PROGRAM MAIN
VAR
	instFB_DryingSectionLubrificationControl_V1 : FB_DryingSectionLubrificationControl_V1;
	instFB_SavePersistentData	: FB_SavePersistentData;
	instFB_SpeedDroopControlMst : FB_SpeedDroopControl_1;
	instFB_SpeedDroopControlSlv : FB_FormingBoardDriveControl;
	instFB_DryingSectionDriveControl_GR1 : FB_DryingSectionDriveControl_V1;
	instFB_DryingSectionDriveControl_GR2 : FB_DryingSectionDriveControl_V1;
	
	instFFB_PressSectionDriveControl_V1 : FB_PressSectionDriveControl_V2;

	                 

	FB_SoftstarterWithBypass_0: FB_SoftstarterWithBypass;
	FB_PressureControl_0: FB_PressureControl;
	FB_MixPumpControl_0: FB_MixPumpControl;
	FB_HeadboxLipsPWMControl_0: FB_HeadboxLipsPWMControl;
	instPWM: CTRL_PWM;
	instFB_MixPumpControl: FB_MixPumpControl;
	instFB_FormingBoardRollUpDown: FB_FormingBoardRollUpDown;
	instFB_HeadboxLipsPWMControl: FB_HeadboxLipsPWMControl;
	instFB_FormingBoarWireStrech: FB_FormingBoardRollUpDown;
	instFB_FormingBoardWireStretchControl: FB_FormingBoardWireStretchControl;
	instFB_SoftstarterSimpleCPS: FB_SimpleMotorStart_V2;
	// Centrifugal Pressure Screen (CPS) running (Depurador cabeçeira)
	CPSRunning: BOOL;
	instFB_LevelControlWirePit: FB_LevelControl_V2;
	instFB_LevelControlCouchPit: FB_LevelControl_V2;
	stop: BOOL;
	formingBoardWireLimitInibit: BOOL;
	instFB_SoftstarterSimpleCouchPitMixer: FB_SimpleMotorStart_V2;
	instFB_SoftstarterWithBypassFormingBoard: FB_SoftstarterWithBypass;
	instFB_SoftstarterWithBypassSuctionRoll: FB_SoftstarterWithBypass_V1;
	FB_SoftstarterWithBypassTest: FB_SoftstarterWithBypass;
	FB_SimpleMotorStart_V2_Test: FB_SimpleMotorStart_V2;
	instFB_SoftstarterWithBypass_V1: FB_SoftstarterWithBypass_V1;
	instFB_PressureControl_V1StockPumpC: FB_PressureControl_V1;
	instFB_SoftstarterWithBypass_FormingBoard: FB_SoftstarterWithBypass_V1;
	instFB_PressureControl_V1: FB_PressureControl_V1;
	instFB_FormingBoardDriveControl_V1: FB_FormingBoardControl_V1;
	instFB_MixPumpControl_V1: FB_MixPumpControl_V1;
	instFB_ProcessControlerStockPump: FB_ProcessControler;
	instFB_ProcessControlerWirePitPump: FB_ProcessControler;
	
	formingBoardNextGrReference: REAL;
	pressSectionNextGrReference: REAL;
	dryingSec1NextGrReference: REAL;
	dryingSec2NextGrReference: REAL;
	
	instFB_DryingSectionDriveControl_GR3: FB_DryingSectionDriveControl_V1;
	
	instFB_DryingSectionDriveControlV2_GR3: FB_DryingSectionDriveControl_V2;
	
	
	
	instFB_RewinderControl_V1 : FB_RewinderControl_V1;
	
	
	
	instFB_DryingSectionDriveControl_V3_GR1: FB_DryingSectionDriveControl_V3;
	instFB_DryingSectionDriveControl_V3_GR2: FB_DryingSectionDriveControl_V3;
	instFB_DryingSectionDriveControl_V3_GR3: FB_DryingSectionDriveControl_V3;
	
	
	initVariables : BOOL;
	rInitVariables : BOOL;
	initVariablesOld : BOOL;
	
	
	dryingSectionGr1NextGroupReference: REAL;
	dryingSectionGr2NextGroupReference: REAL;
	dryingSectionGr3NextGroupReference: REAL;
	instFB_SoftstarterWithBypassPress1: FB_SoftstarterWithBypass_V1;
	instFB_SoftstarterWithBypassPress2: FB_SoftstarterWithBypass_V1;
	bypassFault: BOOL;
	startNotAllowed: BOOL;
	instFB_WinderDriveControl_V1: FB_WinderDriveControl_V1;
	FB_FormingBoardControl_V3_0: FB_FormingBoardControl_V3;
	pressSectionNextGroupReference: REAL;
	
	
	firstScan	:BOOL := TRUE;
	
	
	vacumPumpSoftStartOK: BOOL;
	instTOFvacumPumpSoftstart: TOF;
	startSoftstartContactorFromPressFelt1: BOOL;
	startSoftstartFromPressFelt1: BOOL;
	startSoftstartContactorFromPressFelt2: BOOL;
	startSoftstartFromPressFelt2: BOOL;
	instFB_FB_SimpleMotorStart_V3_VaccumSealPump: FB_SimpleMotorStart_V3;
	instFB_FB_SimpleMotorStart_V3_lowVacuumExhaustFan: FB_SimpleMotorStart_V3;
	instFB_FB_SimpleMotorStart_V3_VaccumSeparator: FB_SimpleMotorStart_V3;
	instFB_FB_SimpleMotorStart_V3_FormingTailCutterNozzle: FB_SimpleMotorStart_V3;
	instFB_FB_SimpleMotorStart_V3_FormingWireShower: FB_SimpleMotorStart_V3;
	
	instFB_AlarmControl	: FB_AlarmControl;
	
END_VAR

//────────────────────────────────────────────
// READ I/O MODULES
//────────────────────────────────────────────

// UG I/O Modules
P1_100_UG01();
P1_100_UG02();
P1_100_UG03_SuctionRoll();
P1_100_UG04();
P1_100_UG05();
P1_300_UG06_TractionRoll();

// Digital Inputs
P1_050_DI1();
P1_050_DI2();
P1_050_DI3();
P9_050_DI1();
P9_050_DI2();
P9_050_DI3();
P10_050_DI1();
P10_050_DI2();
P10_050_DI3();
P10_050_DI4();
P10_050_DI5();
P10_050_DI6();
P10_050_DI7();
P10_050_DI8();

// Digital Outputs
P1_050_DO1();
P1_050_DO2();
P1_050_DO3();
P9_050_DO1();
P9_050_DO2();
P9_050_DO3();
P10_050_DO1();
P10_050_DO2();
P10_050_DO3();
P10_050_DO4();

// Analog Inputs
P1_050_AI1();
P1_050_AI2();
P1_050_AI3();
P1_050_AI4();
P9_050_AI1();
P10_050_AI1();
P10_050_AI2();

// Analog Outputs
P1_050_AQ1();
P1_050_AQ2();
P10_050_AO1();


CP1_050_DI1();
CP1_050_DO1();
CP1_050_AO1();


// Safety PLC
P1_050_SP1();

//────────────────────────────────────────────
// READ DRIVES
//────────────────────────────────────────────

// Press Section
P11_400_UG01_SecondPress();     // Second Press
P12_400_UG01_FirstPress();      // First Press

// Drying Section — Group 1
P13_500_UG01_1GR_UpperSlave();  // Group 1 - Upper Slave
P13_500_UG02_1GR_LowerMaster(); // Group 1 - Lower Master
P13_500_UG03_1GR_UpperMaster(); // Group 1 - Upper Master

// Drying Section — Group 2
P13_501_UG01_2GR_LowerSlave();  // Group 2 - Lower Slave
P13_501_UG02_2GR_UpperSlave();  // Group 2 - Upper Slave
P13_501_UG03_2GR_LowerMaster(); // Group 2 - Lower Master
P14_501_UG01_2GR_UpperMaster(); // Group 2 - Upper Master

// Drying Section — Group 3
P14_502_UG01_3GR_LowerSlave();  // Group 3 - Lower Slave
P14_502_UG02_3GR_UpperSlave();  // Group 3 - Upper Slave
P14_502_UG03_3GR_LowerMaster(); // Group 3 - Lower Master
P14_502_UG04_3GR_UpperMaster(); // Group 3 - Upper Master

//Winder group
P15_600_UG01_Rewinder();
//────────────────────────────────────────────
// PROGRAM FUNCTION BLOCK CALLS
//────────────────────────────────────────────

// Forming Section
_100_FormingBoardControl();
_110_FormingBoardAux();

// Press Section
_200_PressSectionControl();

// Drying Section
_500_DryingSectionGroup1DriveControl();
_501_DryingSectionGroup2DriveControl();
_502_DryingSectionGroup3DriveControl();
_550_DryingSectionLubrification();
_600_WinderGroup();

_888_Alarms();


// Headbox / Stock Prep / Wet End Auxiliary Systems
//_HeadBoxAuxiliaryControls();
_MixPumpControl_1();
_WirePitPumpControl_1();
_CentrifugalPressureScreenControl();
_CouchPitPumpControl();
_CouchPitMixerControl();
_VaccumPumps();
//_StockPumpControl();
_StockPumpControl_1();

// Testing & Debug
_FunctionBlockTest();

//────────────────────────────────────────────
// SYSTEM MANAGEMENT
//────────────────────────────────────────────

// Save persistent variables to CPU
instFB_SavePersistentData();

// Enable Safety PLC
P1_050_SP1.run := TRUE;

// Perform machine-wide reset
machineReset();


rInitVariables := initVariables AND NOT initVariablesOld;

IF rInitVariables THEN
	
	_000_Init_Variables();

END_IF

initVariablesOld := initVariables;



IF firstScan THEN
	
	_001_FirstScan();

END_IF

METHOD _000_Init_Variables
VAR_INPUT
END_VAR

P1_300_UG06_TractionRoll.deviceConfig.MotorSpeedInputLow := 0.0;
P1_300_UG06_TractionRoll.deviceConfig.MotorSpeedInputHigh := 360.4;
P1_300_UG06_TractionRoll.deviceConfig.MotorSpeedOutputLow := 0.0;
P1_300_UG06_TractionRoll.deviceConfig.MotorSpeedOutputHigh := 360.4;
P1_300_UG06_TractionRoll.deviceConfig.speedSetpointInputLow := 0.0;
P1_300_UG06_TractionRoll.deviceConfig.speedSetpointInputHigh := 360.4;
P1_300_UG06_TractionRoll.deviceConfig.speedSetpointOutputLow := 0.0;
P1_300_UG06_TractionRoll.deviceConfig.speedSetpointOutputHigh := 360.4;


P1_100_UG03_SuctionRoll.deviceConfig.MotorSpeedInputLow := 0.0;
P1_100_UG03_SuctionRoll.deviceConfig.MotorSpeedInputHigh := 329.3;
P1_100_UG03_SuctionRoll.deviceConfig.MotorSpeedOutputLow := 0.0;
P1_100_UG03_SuctionRoll.deviceConfig.MotorSpeedOutputHigh := 329.3;
P1_100_UG03_SuctionRoll.deviceConfig.speedSetpointInputLow := 0.0;
P1_100_UG03_SuctionRoll.deviceConfig.speedSetpointInputHigh := 329.3;
P1_100_UG03_SuctionRoll.deviceConfig.speedSetpointOutputLow := 0.0;
P1_100_UG03_SuctionRoll.deviceConfig.speedSetpointOutputHigh := 329.3;
//Torque Enable
P1_100_UG03_SuctionRoll.deviceConfig.torqueLimiterEnabled := TRUE;
P1_100_UG03_SuctionRoll.deviceConfig.operationMode := 4;



P11_400_UG01_SecondPress.deviceConfig.MotorSpeedInputLow := 0.0;
P11_400_UG01_SecondPress.deviceConfig.MotorSpeedInputHigh := 374;
P11_400_UG01_SecondPress.deviceConfig.MotorSpeedOutputLow := 0.0;
P11_400_UG01_SecondPress.deviceConfig.MotorSpeedOutputHigh := 374;
P11_400_UG01_SecondPress.deviceConfig.speedSetpointInputLow := 0.0;
P11_400_UG01_SecondPress.deviceConfig.speedSetpointInputHigh := 374;
P11_400_UG01_SecondPress.deviceConfig.speedSetpointOutputLow := 0.0;
P11_400_UG01_SecondPress.deviceConfig.speedSetpointOutputHigh := 374;


P12_400_UG01_FirstPress.deviceConfig.MotorSpeedInputLow := 0.0;
P12_400_UG01_FirstPress.deviceConfig.MotorSpeedInputHigh := 239.9;
P12_400_UG01_FirstPress.deviceConfig.MotorSpeedOutputLow := 0.0;
P12_400_UG01_FirstPress.deviceConfig.MotorSpeedOutputHigh := 239.9;
P12_400_UG01_FirstPress.deviceConfig.speedSetpointInputLow := 0.0;
P12_400_UG01_FirstPress.deviceConfig.speedSetpointInputHigh := 239.9;
P12_400_UG01_FirstPress.deviceConfig.speedSetpointOutputLow := 0.0;
P12_400_UG01_FirstPress.deviceConfig.speedSetpointOutputHigh := 239.9;
//Torque Enable
P12_400_UG01_FirstPress.deviceConfig.torqueLimiterEnabled := TRUE;
P12_400_UG01_FirstPress.deviceConfig.operationMode := 4;



//============================
// DRYING SECTION — GROUP 1
//============================

// Upper Slave
P13_500_UG01_1GR_UpperSlave.deviceConfig.MotorSpeedInputLow := 0.0;
P13_500_UG01_1GR_UpperSlave.deviceConfig.MotorSpeedInputHigh := 750;
P13_500_UG01_1GR_UpperSlave.deviceConfig.MotorSpeedOutputLow := 0.0;
P13_500_UG01_1GR_UpperSlave.deviceConfig.MotorSpeedOutputHigh := 750;
P13_500_UG01_1GR_UpperSlave.deviceConfig.speedSetpointInputLow := 0.0;
P13_500_UG01_1GR_UpperSlave.deviceConfig.speedSetpointInputHigh := 750;
P13_500_UG01_1GR_UpperSlave.deviceConfig.speedSetpointOutputLow := 0.0;
P13_500_UG01_1GR_UpperSlave.deviceConfig.speedSetpointOutputHigh := 750;
P13_500_UG01_1GR_UpperSlave.deviceConfig.torqueLimiterEnabled := TRUE;
P13_500_UG01_1GR_UpperSlave.deviceConfig.operationMode := 4;

// Lower Master
P13_500_UG02_1GR_LowerMaster.deviceConfig.MotorSpeedInputLow := 0.0;
P13_500_UG02_1GR_LowerMaster.deviceConfig.MotorSpeedInputHigh := 750;
P13_500_UG02_1GR_LowerMaster.deviceConfig.MotorSpeedOutputLow := 0.0;
P13_500_UG02_1GR_LowerMaster.deviceConfig.MotorSpeedOutputHigh := 750;
P13_500_UG02_1GR_LowerMaster.deviceConfig.speedSetpointInputLow := 0.0;
P13_500_UG02_1GR_LowerMaster.deviceConfig.speedSetpointInputHigh := 750;
P13_500_UG02_1GR_LowerMaster.deviceConfig.speedSetpointOutputLow := 0.0;
P13_500_UG02_1GR_LowerMaster.deviceConfig.speedSetpointOutputHigh := 750;
//P13_500_UG02_1GR_LowerMaster.deviceConfig.torqueLimiterEnabled := FALSE;
//P13_500_UG02_1GR_LowerMaster.deviceConfig.operationMode := 4;

// Upper Master
P13_500_UG03_1GR_UpperMaster.deviceConfig.MotorSpeedInputLow := 0.0;
P13_500_UG03_1GR_UpperMaster.deviceConfig.MotorSpeedInputHigh := 750;
P13_500_UG03_1GR_UpperMaster.deviceConfig.MotorSpeedOutputLow := 0.0;
P13_500_UG03_1GR_UpperMaster.deviceConfig.MotorSpeedOutputHigh := 750;
P13_500_UG03_1GR_UpperMaster.deviceConfig.speedSetpointInputLow := 0.0;
P13_500_UG03_1GR_UpperMaster.deviceConfig.speedSetpointInputHigh := 750;
P13_500_UG03_1GR_UpperMaster.deviceConfig.speedSetpointOutputLow := 0.0;
P13_500_UG03_1GR_UpperMaster.deviceConfig.speedSetpointOutputHigh := 750;
//P13_500_UG03_1GR_UpperMaster.deviceConfig.torqueLimiterEnabled := FALSE;
//P13_500_UG03_1GR_UpperMaster.deviceConfig.operationMode := 4;


//============================
// DRYING SECTION — GROUP 2
//============================

// Lower Slave
P13_501_UG01_2GR_LowerSlave.deviceConfig.MotorSpeedInputLow := 0.0;
P13_501_UG01_2GR_LowerSlave.deviceConfig.MotorSpeedInputHigh := 750;
P13_501_UG01_2GR_LowerSlave.deviceConfig.MotorSpeedOutputLow := 0.0;
P13_501_UG01_2GR_LowerSlave.deviceConfig.MotorSpeedOutputHigh := 750;
P13_501_UG01_2GR_LowerSlave.deviceConfig.speedSetpointInputLow := 0.0;
P13_501_UG01_2GR_LowerSlave.deviceConfig.speedSetpointInputHigh := 750;
P13_501_UG01_2GR_LowerSlave.deviceConfig.speedSetpointOutputLow := 0.0;
P13_501_UG01_2GR_LowerSlave.deviceConfig.speedSetpointOutputHigh := 750;
P13_501_UG01_2GR_LowerSlave.deviceConfig.torqueLimiterEnabled := TRUE;
P13_501_UG01_2GR_LowerSlave.deviceConfig.operationMode := 4;

// Upper Slave
P13_501_UG02_2GR_UpperSlave.deviceConfig.MotorSpeedInputLow := 0.0;
P13_501_UG02_2GR_UpperSlave.deviceConfig.MotorSpeedInputHigh := 750;
P13_501_UG02_2GR_UpperSlave.deviceConfig.MotorSpeedOutputLow := 0.0;
P13_501_UG02_2GR_UpperSlave.deviceConfig.MotorSpeedOutputHigh := 750;
P13_501_UG02_2GR_UpperSlave.deviceConfig.speedSetpointInputLow := 0.0;
P13_501_UG02_2GR_UpperSlave.deviceConfig.speedSetpointInputHigh := 750;
P13_501_UG02_2GR_UpperSlave.deviceConfig.speedSetpointOutputLow := 0.0;
P13_501_UG02_2GR_UpperSlave.deviceConfig.speedSetpointOutputHigh := 750;
P13_501_UG02_2GR_UpperSlave.deviceConfig.torqueLimiterEnabled := TRUE;
P13_501_UG02_2GR_UpperSlave.deviceConfig.operationMode := 4;

// Lower Master
P13_501_UG03_2GR_LowerMaster.deviceConfig.MotorSpeedInputLow := 0.0;
P13_501_UG03_2GR_LowerMaster.deviceConfig.MotorSpeedInputHigh := 750;
P13_501_UG03_2GR_LowerMaster.deviceConfig.MotorSpeedOutputLow := 0.0;
P13_501_UG03_2GR_LowerMaster.deviceConfig.MotorSpeedOutputHigh := 750;
P13_501_UG03_2GR_LowerMaster.deviceConfig.speedSetpointInputLow := 0.0;
P13_501_UG03_2GR_LowerMaster.deviceConfig.speedSetpointInputHigh := 750;
P13_501_UG03_2GR_LowerMaster.deviceConfig.speedSetpointOutputLow := 0.0;
P13_501_UG03_2GR_LowerMaster.deviceConfig.speedSetpointOutputHigh := 750;
//P13_501_UG03_2GR_LowerMaster.deviceConfig.torqueLimiterEnabled := FALSE;
//P13_501_UG03_2GR_LowerMaster.deviceConfig.operationMode := 4;

// Upper Master
P14_501_UG01_2GR_UpperMaster.deviceConfig.MotorSpeedInputLow := 0.0;
P14_501_UG01_2GR_UpperMaster.deviceConfig.MotorSpeedInputHigh := 750;
P14_501_UG01_2GR_UpperMaster.deviceConfig.MotorSpeedOutputLow := 0.0;
P14_501_UG01_2GR_UpperMaster.deviceConfig.MotorSpeedOutputHigh := 750;
P14_501_UG01_2GR_UpperMaster.deviceConfig.speedSetpointInputLow := 0.0;
P14_501_UG01_2GR_UpperMaster.deviceConfig.speedSetpointInputHigh := 750;
P14_501_UG01_2GR_UpperMaster.deviceConfig.speedSetpointOutputLow := 0.0;
P14_501_UG01_2GR_UpperMaster.deviceConfig.speedSetpointOutputHigh := 750;
//P14_501_UG01_2GR_UpperMaster.deviceConfig.torqueLimiterEnabled := FALSE;
//P14_501_UG01_2GR_UpperMaster.deviceConfig.operationMode := 4;


//============================
// DRYING SECTION — GROUP 3
//============================

// Lower Slave
P14_502_UG01_3GR_LowerSlave.deviceConfig.MotorSpeedInputLow := 0.0;
P14_502_UG01_3GR_LowerSlave.deviceConfig.MotorSpeedInputHigh := 750;
P14_502_UG01_3GR_LowerSlave.deviceConfig.MotorSpeedOutputLow := 0.0;
P14_502_UG01_3GR_LowerSlave.deviceConfig.MotorSpeedOutputHigh := 750;
P14_502_UG01_3GR_LowerSlave.deviceConfig.speedSetpointInputLow := 0.0;
P14_502_UG01_3GR_LowerSlave.deviceConfig.speedSetpointInputHigh := 750;
P14_502_UG01_3GR_LowerSlave.deviceConfig.speedSetpointOutputLow := 0.0;
P14_502_UG01_3GR_LowerSlave.deviceConfig.speedSetpointOutputHigh := 750;
P14_502_UG01_3GR_LowerSlave.deviceConfig.torqueLimiterEnabled := TRUE;
P14_502_UG01_3GR_LowerSlave.deviceConfig.operationMode := 4;

// Upper Slave
P14_502_UG02_3GR_UpperSlave.deviceConfig.MotorSpeedInputLow := 0.0;
P14_502_UG02_3GR_UpperSlave.deviceConfig.MotorSpeedInputHigh := 750;
P14_502_UG02_3GR_UpperSlave.deviceConfig.MotorSpeedOutputLow := 0.0;
P14_502_UG02_3GR_UpperSlave.deviceConfig.MotorSpeedOutputHigh := 750;
P14_502_UG02_3GR_UpperSlave.deviceConfig.speedSetpointInputLow := 0.0;
P14_502_UG02_3GR_UpperSlave.deviceConfig.speedSetpointInputHigh := 750;
P14_502_UG02_3GR_UpperSlave.deviceConfig.speedSetpointOutputLow := 0.0;
P14_502_UG02_3GR_UpperSlave.deviceConfig.speedSetpointOutputHigh := 750;
P14_502_UG02_3GR_UpperSlave.deviceConfig.torqueLimiterEnabled := TRUE;
P14_502_UG02_3GR_UpperSlave.deviceConfig.operationMode := 4;

// Lower Master
P14_502_UG03_3GR_LowerMaster.deviceConfig.MotorSpeedInputLow := 0.0;
P14_502_UG03_3GR_LowerMaster.deviceConfig.MotorSpeedInputHigh := 750;
P14_502_UG03_3GR_LowerMaster.deviceConfig.MotorSpeedOutputLow := 0.0;
P14_502_UG03_3GR_LowerMaster.deviceConfig.MotorSpeedOutputHigh := 750;
P14_502_UG03_3GR_LowerMaster.deviceConfig.speedSetpointInputLow := 0.0;
P14_502_UG03_3GR_LowerMaster.deviceConfig.speedSetpointInputHigh := 750;
P14_502_UG03_3GR_LowerMaster.deviceConfig.speedSetpointOutputLow := 0.0;
P14_502_UG03_3GR_LowerMaster.deviceConfig.speedSetpointOutputHigh := 750;
//P14_502_UG03_3GR_LowerMaster.deviceConfig.torqueLimiterEnabled := FALSE;
//P14_502_UG03_3GR_LowerMaster.deviceConfig.operationMode := 4;

// Upper Master
P14_502_UG04_3GR_UpperMaster.deviceConfig.MotorSpeedInputLow := 0.0;
P14_502_UG04_3GR_UpperMaster.deviceConfig.MotorSpeedInputHigh := 750;
P14_502_UG04_3GR_UpperMaster.deviceConfig.MotorSpeedOutputLow := 0.0;
P14_502_UG04_3GR_UpperMaster.deviceConfig.MotorSpeedOutputHigh := 750;
P14_502_UG04_3GR_UpperMaster.deviceConfig.speedSetpointInputLow := 0.0;
P14_502_UG04_3GR_UpperMaster.deviceConfig.speedSetpointInputHigh := 750;
P14_502_UG04_3GR_UpperMaster.deviceConfig.speedSetpointOutputLow := 0.0;
P14_502_UG04_3GR_UpperMaster.deviceConfig.speedSetpointOutputHigh := 750;
//P14_502_UG04_3GR_UpperMaster.deviceConfig.torqueLimiterEnabled := FALSE;
//P14_502_UG04_3GR_UpperMaster.deviceConfig.operationMode := 4;
END_METHOD

METHOD _001_FirstScan
VAR_INPUT
END_VAR

(*

paperMachineHmiCommands.dryingSectionGroup1SteamPressureAutoMan := FALSE;

	dryingSectionGroup1SteamPressureAutoSetpoint : REAL;  // Recovery speed increment [m/min or %] (Incremento de recuperação Grupo 1)
	dryingSectionGroup1SteamPressureManualSetpoint : REAL;  // Recovery speed increment [m/min or %] (Incremento de recuperação Grupo 1)
	
*)



paperMachineHmiCommands.dryingSectionGroup1SteamPressureAutoMan := FALSE;
paperMachineHmiCommands.dryingSectionGroup1SteamPressureManualSetpoint := 0.0;

paperMachineHmiCommands.dryingSectionGroup2SteamPressureAutoMan := FALSE;
paperMachineHmiCommands.dryingSectionGroup2SteamPressureManualSetpoint := 0.0;

paperMachineHmiCommands.dryingSectionGroup3SteamPressureAutoMan := FALSE;
paperMachineHmiCommands.dryingSectionGroup3SteamPressureManualSetpoint := 0.0;


//Reset first scan flag
firstScan := FALSE;
END_METHOD

METHOD _100_FormingBoardControl
VAR_INPUT
END_VAR
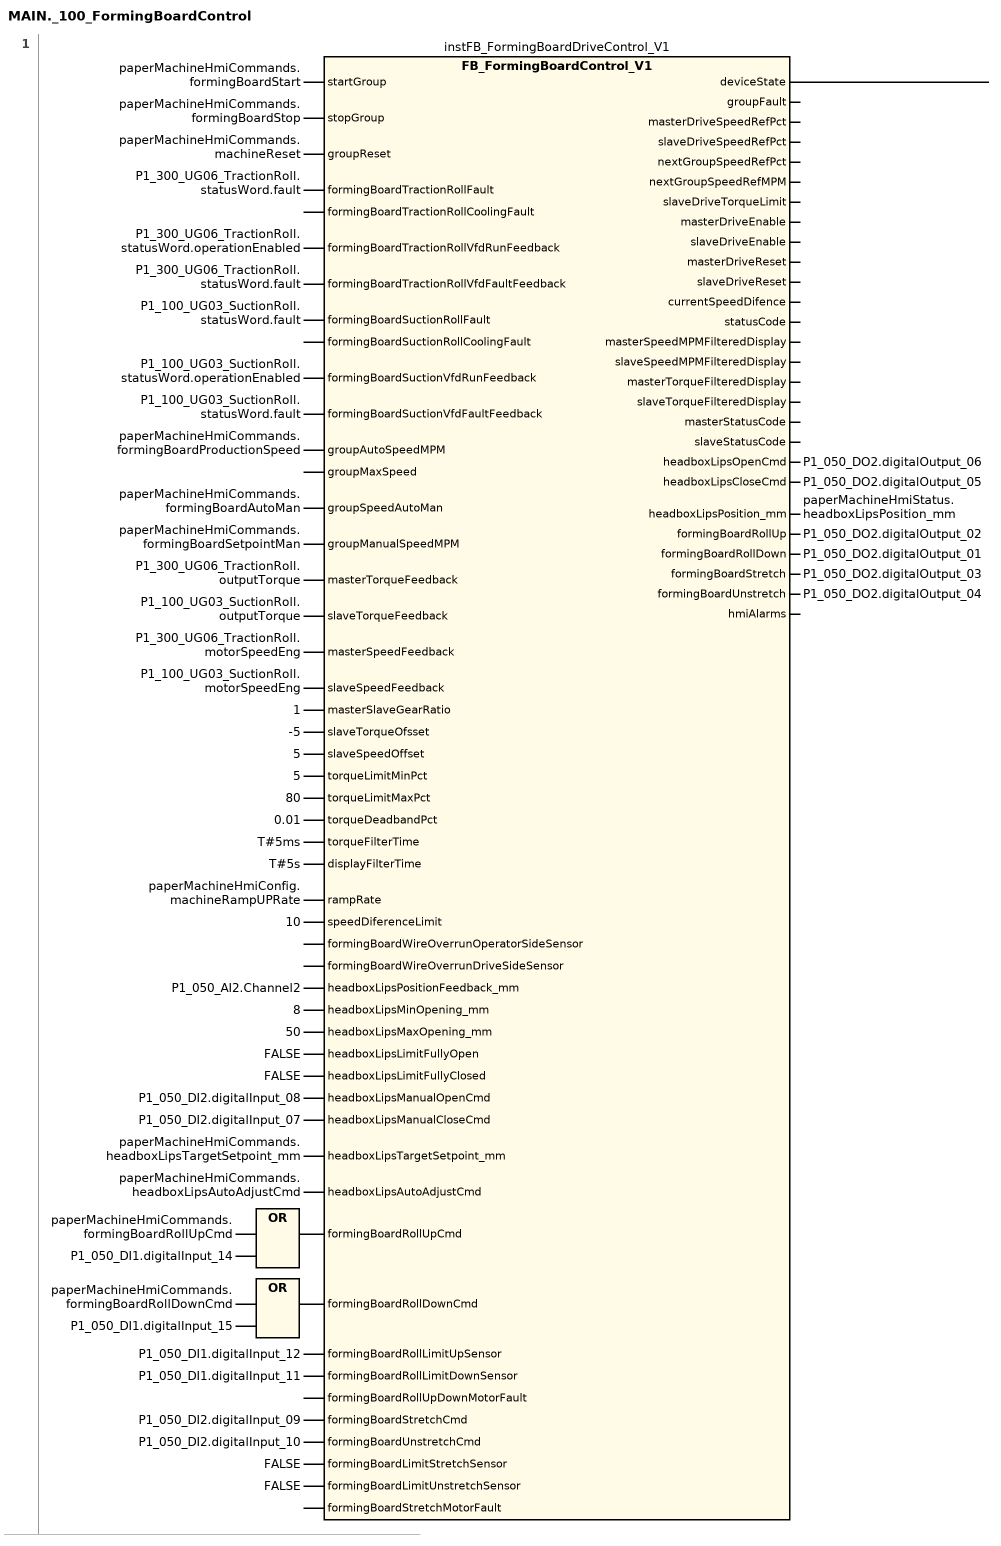
// NETWORK 1
instFB_FormingBoardDriveControl_V1(
    startGroup := paperMachineHmiCommands.formingBoardStart,
    stopGroup := paperMachineHmiCommands.formingBoardStop,
    groupReset := paperMachineHmiCommands.machineReset,
    formingBoardTractionRollFault := P1_300_UG06_TractionRoll.statusWord.fault,
    formingBoardTractionRollVfdRunFeedback := P1_300_UG06_TractionRoll.statusWord.operationEnabled,
    formingBoardTractionRollVfdFaultFeedback := P1_300_UG06_TractionRoll.statusWord.fault,
    formingBoardSuctionRollFault := P1_100_UG03_SuctionRoll.statusWord.fault,
    formingBoardSuctionVfdRunFeedback := P1_100_UG03_SuctionRoll.statusWord.operationEnabled,
    formingBoardSuctionVfdFaultFeedback := P1_100_UG03_SuctionRoll.statusWord.fault,
    groupAutoSpeedMPM := paperMachineHmiCommands.formingBoardProductionSpeed,
    groupSpeedAutoMan := paperMachineHmiCommands.formingBoardAutoMan,
    groupManualSpeedMPM := paperMachineHmiCommands.formingBoardSetpointMan,
    masterTorqueFeedback := P1_300_UG06_TractionRoll.outputTorque,
    slaveTorqueFeedback := P1_100_UG03_SuctionRoll.outputTorque,
    masterSpeedFeedback := P1_300_UG06_TractionRoll.motorSpeedEng,
    slaveSpeedFeedback := P1_100_UG03_SuctionRoll.motorSpeedEng,
    masterSlaveGearRatio := 1,
    slaveTorqueOfsset := -5,
    slaveSpeedOffset := 5,
    torqueLimitMinPct := 5,
    torqueLimitMaxPct := 80,
    torqueDeadbandPct := 0.01,
    torqueFilterTime := T#5ms,
    displayFilterTime := T#5s,
    rampRate := paperMachineHmiConfig.machineRampUPRate,
    speedDiferenceLimit := 10,
    headboxLipsPositionFeedback_mm := P1_050_AI2.Channel2,
    headboxLipsMinOpening_mm := 8,
    headboxLipsMaxOpening_mm := 50,
    headboxLipsLimitFullyOpen := FALSE,
    headboxLipsLimitFullyClosed := FALSE,
    headboxLipsManualOpenCmd := P1_050_DI2.digitalInput_08,
    headboxLipsManualCloseCmd := P1_050_DI2.digitalInput_07,
    headboxLipsTargetSetpoint_mm := paperMachineHmiCommands.headboxLipsTargetSetpoint_mm,
    headboxLipsAutoAdjustCmd := paperMachineHmiCommands.headboxLipsAutoAdjustCmd,
    formingBoardRollUpCmd := paperMachineHmiCommands.formingBoardRollUpCmd OR P1_050_DI1.digitalInput_14,
    formingBoardRollDownCmd := paperMachineHmiCommands.formingBoardRollDownCmd OR P1_050_DI1.digitalInput_15,
    formingBoardRollLimitUpSensor := P1_050_DI1.digitalInput_12,
    formingBoardRollLimitDownSensor := P1_050_DI1.digitalInput_11,
    formingBoardStretchCmd := P1_050_DI2.digitalInput_09,
    formingBoardUnstretchCmd := P1_050_DI2.digitalInput_10,
    formingBoardLimitStretchSensor := FALSE,
    formingBoardLimitUnstretchSensor := FALSE,
    headboxLipsOpenCmd => P1_050_DO2.digitalOutput_06,
    headboxLipsCloseCmd => P1_050_DO2.digitalOutput_05,
    headboxLipsPosition_mm => paperMachineHmiStatus.headboxLipsPosition_mm,
    formingBoardRollUp => P1_050_DO2.digitalOutput_02,
    formingBoardRollDown => P1_050_DO2.digitalOutput_01,
    formingBoardStretch => P1_050_DO2.digitalOutput_03,
    formingBoardUnstretch => P1_050_DO2.digitalOutput_04); // FB_FormingBoardControl_V1

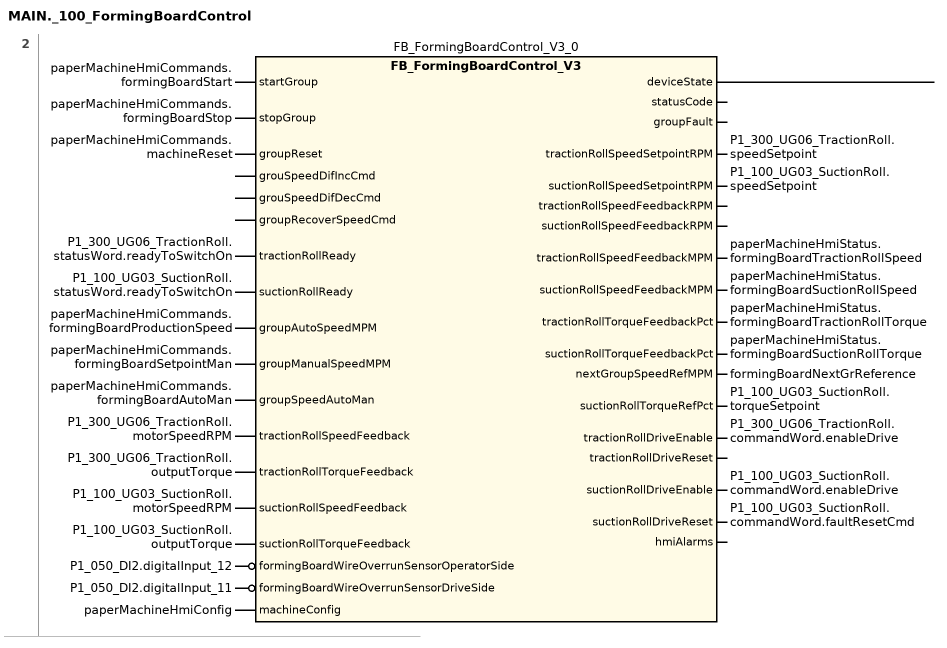
// NETWORK 2
FB_FormingBoardControl_V3_0(
    startGroup := paperMachineHmiCommands.formingBoardStart,
    stopGroup := paperMachineHmiCommands.formingBoardStop,
    groupReset := paperMachineHmiCommands.machineReset,
    tractionRollReady := P1_300_UG06_TractionRoll.statusWord.readyToSwitchOn,
    suctionRollReady := P1_100_UG03_SuctionRoll.statusWord.readyToSwitchOn,
    groupAutoSpeedMPM := paperMachineHmiCommands.formingBoardProductionSpeed,
    groupManualSpeedMPM := paperMachineHmiCommands.formingBoardSetpointMan,
    groupSpeedAutoMan := paperMachineHmiCommands.formingBoardAutoMan,
    tractionRollSpeedFeedback := P1_300_UG06_TractionRoll.motorSpeedRPM,
    tractionRollTorqueFeedback := P1_300_UG06_TractionRoll.outputTorque,
    suctionRollSpeedFeedback := P1_100_UG03_SuctionRoll.motorSpeedRPM,
    suctionRollTorqueFeedback := P1_100_UG03_SuctionRoll.outputTorque,
    formingBoardWireOverrunSensorOperatorSide := NOT P1_050_DI2.digitalInput_12,
    formingBoardWireOverrunSensorDriveSide := NOT P1_050_DI2.digitalInput_11,
    machineConfig := paperMachineHmiConfig,
    tractionRollSpeedSetpointRPM => P1_300_UG06_TractionRoll.speedSetpoint,
    suctionRollSpeedSetpointRPM => P1_100_UG03_SuctionRoll.speedSetpoint,
    tractionRollSpeedFeedbackMPM => paperMachineHmiStatus.formingBoardTractionRollSpeed,
    suctionRollSpeedFeedbackMPM => paperMachineHmiStatus.formingBoardSuctionRollSpeed,
    tractionRollTorqueFeedbackPct => paperMachineHmiStatus.formingBoardTractionRollTorque,
    suctionRollTorqueFeedbackPct => paperMachineHmiStatus.formingBoardSuctionRollTorque,
    nextGroupSpeedRefMPM => formingBoardNextGrReference,
    suctionRollTorqueRefPct => P1_100_UG03_SuctionRoll.torqueSetpoint,
    tractionRollDriveEnable => P1_300_UG06_TractionRoll.commandWord.enableDrive,
    suctionRollDriveEnable => P1_100_UG03_SuctionRoll.commandWord.enableDrive,
    suctionRollDriveReset => P1_100_UG03_SuctionRoll.commandWord.faultResetCmd); // FB_FormingBoardControl_V3
END_METHOD

METHOD _110_FormingBoardAux
VAR_INPUT
END_VAR
(*


	formingTailCutterNozzleStartCmd   : BOOL; 
	formingTailCutterNozzleStopCmd   : BOOL; 
	formingWireShowerStartCmd : BOOL; 
	formingWireShowerStopCmd : BOOL; 	

*)
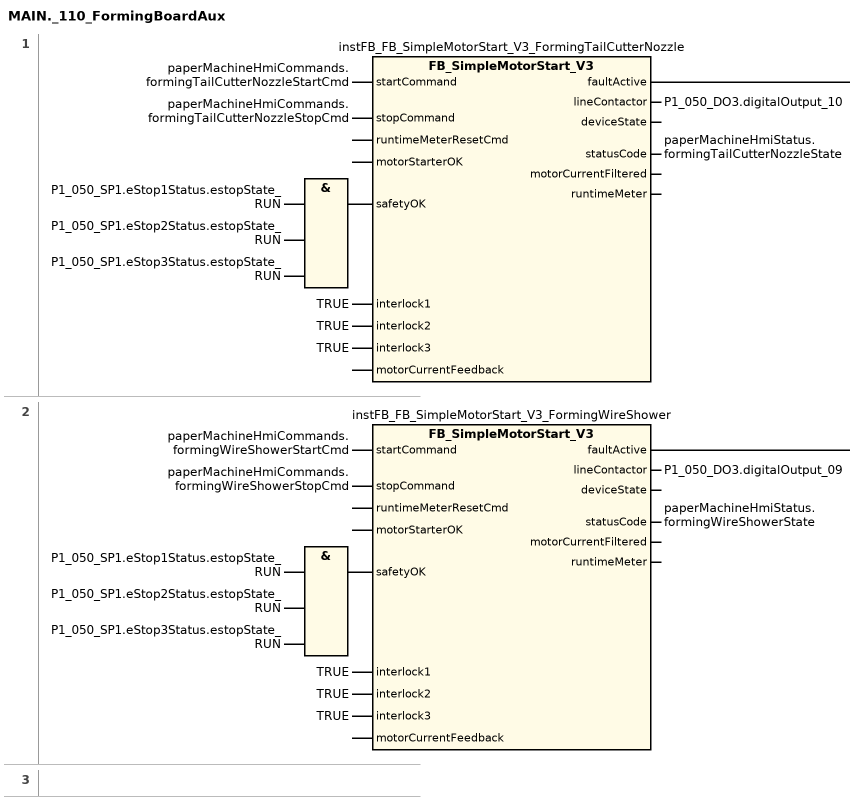
// NETWORK 1
instFB_FB_SimpleMotorStart_V3_FormingTailCutterNozzle(
    startCommand := paperMachineHmiCommands.formingTailCutterNozzleStartCmd,
    stopCommand := paperMachineHmiCommands.formingTailCutterNozzleStopCmd,
    safetyOK := P1_050_SP1.eStop1Status.estopState_RUN AND P1_050_SP1.eStop2Status.estopState_RUN AND P1_050_SP1.eStop3Status.estopState_RUN,
    interlock1 := TRUE,
    interlock2 := TRUE,
    interlock3 := TRUE,
    lineContactor => P1_050_DO3.digitalOutput_10,
    statusCode => paperMachineHmiStatus.formingTailCutterNozzleState); // FB_SimpleMotorStart_V3

// NETWORK 2
instFB_FB_SimpleMotorStart_V3_FormingWireShower(
    startCommand := paperMachineHmiCommands.formingWireShowerStartCmd,
    stopCommand := paperMachineHmiCommands.formingWireShowerStopCmd,
    safetyOK := P1_050_SP1.eStop1Status.estopState_RUN AND P1_050_SP1.eStop2Status.estopState_RUN AND P1_050_SP1.eStop3Status.estopState_RUN,
    interlock1 := TRUE,
    interlock2 := TRUE,
    interlock3 := TRUE,
    lineContactor => P1_050_DO3.digitalOutput_09,
    statusCode => paperMachineHmiStatus.formingWireShowerState); // FB_SimpleMotorStart_V3

// NETWORK 3
END_METHOD

METHOD _200_PressSectionControl
VAR_INPUT
END_VAR
(*

P1_200_UG01();	//First press group master motor
P1_200_UG02();	//First press group slave motor
	
P1_300_UG01();	//First drying group master motor
P1_300_UG02();	//First drying group slave 1
P1_300_UG03();	//First drying group slave 2
	
P1_400_UG01();	//Second drying group master motor
P1_400_UG02();	//Second drying group slave 1
P1_400_UG03();	//Second drying group slave 2

*)
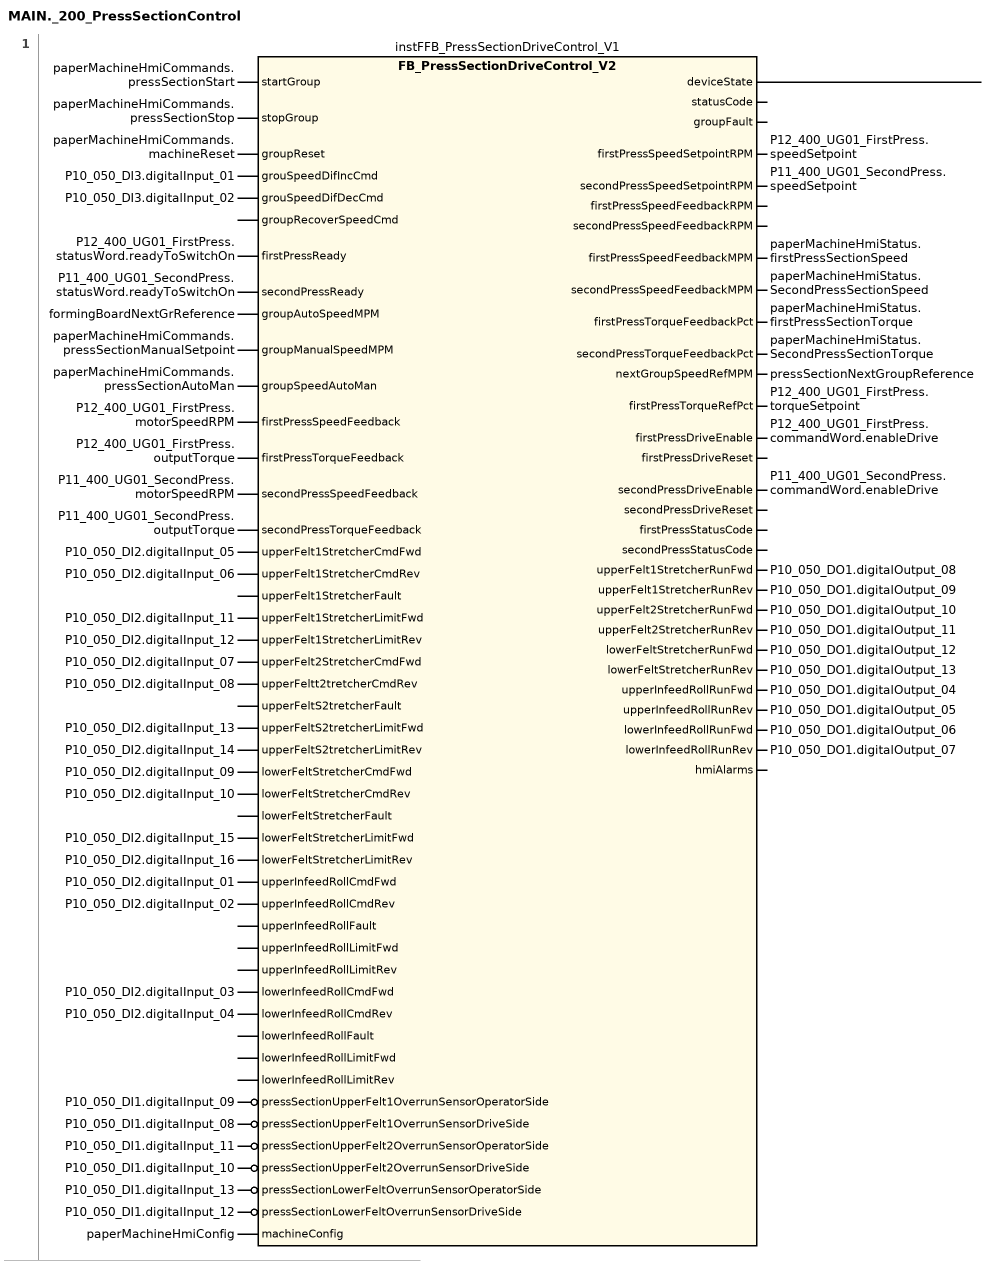
// NETWORK 1
instFFB_PressSectionDriveControl_V1(
    startGroup := paperMachineHmiCommands.pressSectionStart,
    stopGroup := paperMachineHmiCommands.pressSectionStop,
    groupReset := paperMachineHmiCommands.machineReset,
    grouSpeedDifIncCmd := P10_050_DI3.digitalInput_01,
    grouSpeedDifDecCmd := P10_050_DI3.digitalInput_02,
    firstPressReady := P12_400_UG01_FirstPress.statusWord.readyToSwitchOn,
    secondPressReady := P11_400_UG01_SecondPress.statusWord.readyToSwitchOn,
    groupAutoSpeedMPM := formingBoardNextGrReference,
    groupManualSpeedMPM := paperMachineHmiCommands.pressSectionManualSetpoint,
    groupSpeedAutoMan := paperMachineHmiCommands.pressSectionAutoMan,
    firstPressSpeedFeedback := P12_400_UG01_FirstPress.motorSpeedRPM,
    firstPressTorqueFeedback := P12_400_UG01_FirstPress.outputTorque,
    secondPressSpeedFeedback := P11_400_UG01_SecondPress.motorSpeedRPM,
    secondPressTorqueFeedback := P11_400_UG01_SecondPress.outputTorque,
    upperFelt1StretcherCmdFwd := P10_050_DI2.digitalInput_05,
    upperFelt1StretcherCmdRev := P10_050_DI2.digitalInput_06,
    upperFelt1StretcherLimitFwd := P10_050_DI2.digitalInput_11,
    upperFelt1StretcherLimitRev := P10_050_DI2.digitalInput_12,
    upperFelt2StretcherCmdFwd := P10_050_DI2.digitalInput_07,
    upperFeltt2tretcherCmdRev := P10_050_DI2.digitalInput_08,
    upperFeltS2tretcherLimitFwd := P10_050_DI2.digitalInput_13,
    upperFeltS2tretcherLimitRev := P10_050_DI2.digitalInput_14,
    lowerFeltStretcherCmdFwd := P10_050_DI2.digitalInput_09,
    lowerFeltStretcherCmdRev := P10_050_DI2.digitalInput_10,
    lowerFeltStretcherLimitFwd := P10_050_DI2.digitalInput_15,
    lowerFeltStretcherLimitRev := P10_050_DI2.digitalInput_16,
    upperInfeedRollCmdFwd := P10_050_DI2.digitalInput_01,
    upperInfeedRollCmdRev := P10_050_DI2.digitalInput_02,
    lowerInfeedRollCmdFwd := P10_050_DI2.digitalInput_03,
    lowerInfeedRollCmdRev := P10_050_DI2.digitalInput_04,
    pressSectionUpperFelt1OverrunSensorOperatorSide := NOT P10_050_DI1.digitalInput_09,
    pressSectionUpperFelt1OverrunSensorDriveSide := NOT P10_050_DI1.digitalInput_08,
    pressSectionUpperFelt2OverrunSensorOperatorSide := NOT P10_050_DI1.digitalInput_11,
    pressSectionUpperFelt2OverrunSensorDriveSide := NOT P10_050_DI1.digitalInput_10,
    pressSectionLowerFeltOverrunSensorOperatorSide := NOT P10_050_DI1.digitalInput_13,
    pressSectionLowerFeltOverrunSensorDriveSide := NOT P10_050_DI1.digitalInput_12,
    machineConfig := paperMachineHmiConfig,
    firstPressSpeedSetpointRPM => P12_400_UG01_FirstPress.speedSetpoint,
    secondPressSpeedSetpointRPM => P11_400_UG01_SecondPress.speedSetpoint,
    firstPressSpeedFeedbackMPM => paperMachineHmiStatus.firstPressSectionSpeed,
    secondPressSpeedFeedbackMPM => paperMachineHmiStatus.SecondPressSectionSpeed,
    firstPressTorqueFeedbackPct => paperMachineHmiStatus.firstPressSectionTorque,
    secondPressTorqueFeedbackPct => paperMachineHmiStatus.SecondPressSectionTorque,
    nextGroupSpeedRefMPM => pressSectionNextGroupReference,
    firstPressTorqueRefPct => P12_400_UG01_FirstPress.torqueSetpoint,
    firstPressDriveEnable => P12_400_UG01_FirstPress.commandWord.enableDrive,
    secondPressDriveEnable => P11_400_UG01_SecondPress.commandWord.enableDrive,
    upperFelt1StretcherRunFwd => P10_050_DO1.digitalOutput_08,
    upperFelt1StretcherRunRev => P10_050_DO1.digitalOutput_09,
    upperFelt2StretcherRunFwd => P10_050_DO1.digitalOutput_10,
    upperFelt2StretcherRunRev => P10_050_DO1.digitalOutput_11,
    lowerFeltStretcherRunFwd => P10_050_DO1.digitalOutput_12,
    lowerFeltStretcherRunRev => P10_050_DO1.digitalOutput_13,
    upperInfeedRollRunFwd => P10_050_DO1.digitalOutput_04,
    upperInfeedRollRunRev => P10_050_DO1.digitalOutput_05,
    lowerInfeedRollRunFwd => P10_050_DO1.digitalOutput_06,
    lowerInfeedRollRunRev => P10_050_DO1.digitalOutput_07); // FB_PressSectionDriveControl_V2
END_METHOD

METHOD _500_DryingSectionGroup1DriveControl
VAR_INPUT
END_VAR

(*

	dryingSectionGroup1SteamPressureAutoMan : BOOL;  // Recovery speed increment [m/min or %] (Incremento de recuperação Grupo 1)
	dryingSectionGroup1SteamPressureAutoSetpoint : REAL;  // Recovery speed increment [m/min or %] (Incremento de recuperação Grupo 1)
	dryingSectionGroup1SteamPressureManualSetpoint : REAL;  // Recovery speed increment [m/min or %] (Incremento de recuperação Grupo 1)
	
*)
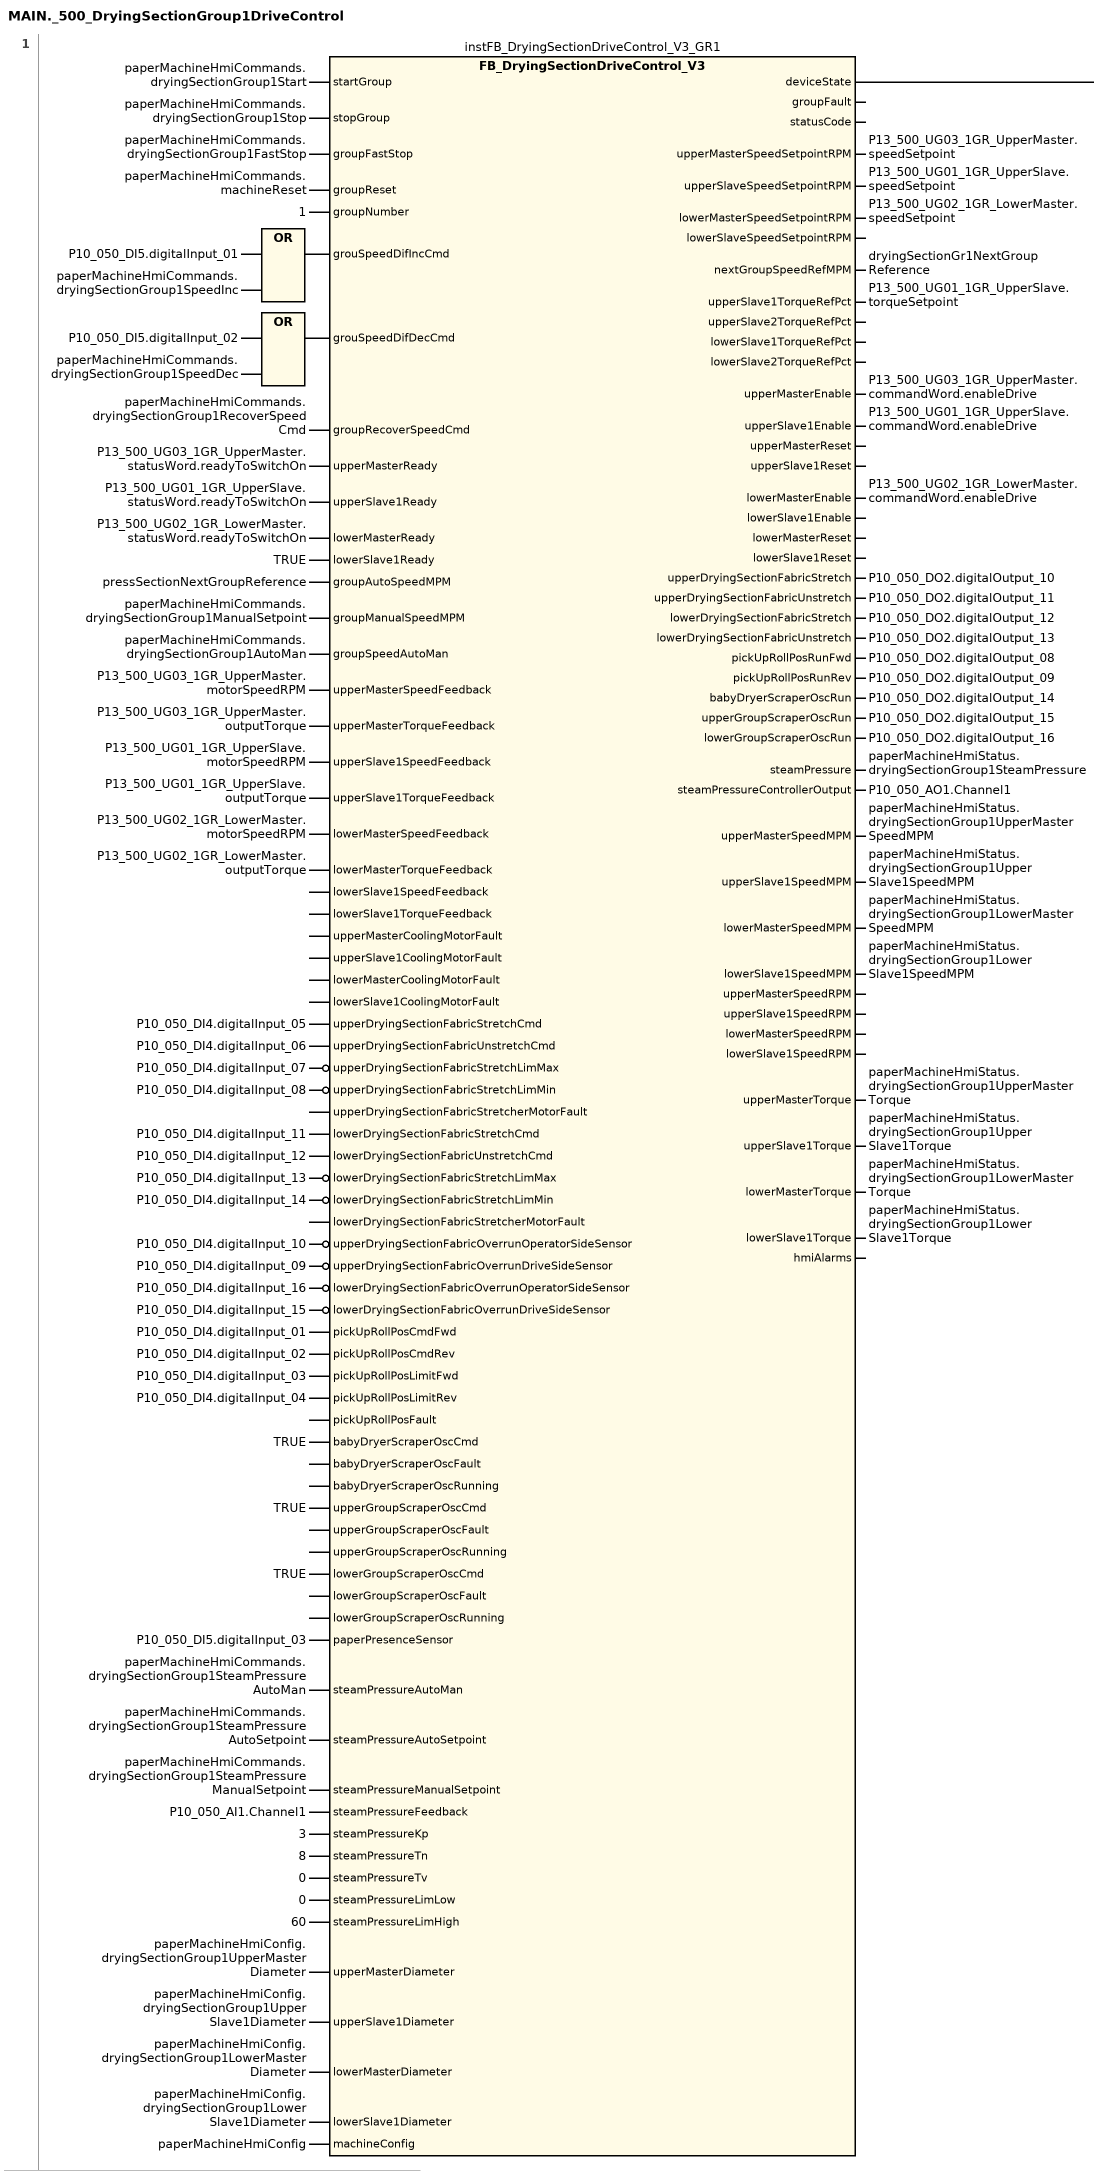
// NETWORK 1
instFB_DryingSectionDriveControl_V3_GR1(
    startGroup := paperMachineHmiCommands.dryingSectionGroup1Start,
    stopGroup := paperMachineHmiCommands.dryingSectionGroup1Stop,
    groupFastStop := paperMachineHmiCommands.dryingSectionGroup1FastStop,
    groupReset := paperMachineHmiCommands.machineReset,
    groupNumber := 1,
    grouSpeedDifIncCmd := P10_050_DI5.digitalInput_01 OR paperMachineHmiCommands.dryingSectionGroup1SpeedInc,
    grouSpeedDifDecCmd := P10_050_DI5.digitalInput_02 OR paperMachineHmiCommands.dryingSectionGroup1SpeedDec,
    groupRecoverSpeedCmd := paperMachineHmiCommands.dryingSectionGroup1RecoverSpeedCmd,
    upperMasterReady := P13_500_UG03_1GR_UpperMaster.statusWord.readyToSwitchOn,
    upperSlave1Ready := P13_500_UG01_1GR_UpperSlave.statusWord.readyToSwitchOn,
    lowerMasterReady := P13_500_UG02_1GR_LowerMaster.statusWord.readyToSwitchOn,
    lowerSlave1Ready := TRUE,
    groupAutoSpeedMPM := pressSectionNextGroupReference,
    groupManualSpeedMPM := paperMachineHmiCommands.dryingSectionGroup1ManualSetpoint,
    groupSpeedAutoMan := paperMachineHmiCommands.dryingSectionGroup1AutoMan,
    upperMasterSpeedFeedback := P13_500_UG03_1GR_UpperMaster.motorSpeedRPM,
    upperMasterTorqueFeedback := P13_500_UG03_1GR_UpperMaster.outputTorque,
    upperSlave1SpeedFeedback := P13_500_UG01_1GR_UpperSlave.motorSpeedRPM,
    upperSlave1TorqueFeedback := P13_500_UG01_1GR_UpperSlave.outputTorque,
    lowerMasterSpeedFeedback := P13_500_UG02_1GR_LowerMaster.motorSpeedRPM,
    lowerMasterTorqueFeedback := P13_500_UG02_1GR_LowerMaster.outputTorque,
    upperDryingSectionFabricStretchCmd := P10_050_DI4.digitalInput_05,
    upperDryingSectionFabricUnstretchCmd := P10_050_DI4.digitalInput_06,
    upperDryingSectionFabricStretchLimMax := NOT P10_050_DI4.digitalInput_07,
    upperDryingSectionFabricStretchLimMin := NOT P10_050_DI4.digitalInput_08,
    lowerDryingSectionFabricStretchCmd := P10_050_DI4.digitalInput_11,
    lowerDryingSectionFabricUnstretchCmd := P10_050_DI4.digitalInput_12,
    lowerDryingSectionFabricStretchLimMax := NOT P10_050_DI4.digitalInput_13,
    lowerDryingSectionFabricStretchLimMin := NOT P10_050_DI4.digitalInput_14,
    upperDryingSectionFabricOverrunOperatorSideSensor := NOT P10_050_DI4.digitalInput_10,
    upperDryingSectionFabricOverrunDriveSideSensor := NOT P10_050_DI4.digitalInput_09,
    lowerDryingSectionFabricOverrunOperatorSideSensor := NOT P10_050_DI4.digitalInput_16,
    lowerDryingSectionFabricOverrunDriveSideSensor := NOT P10_050_DI4.digitalInput_15,
    pickUpRollPosCmdFwd := P10_050_DI4.digitalInput_01,
    pickUpRollPosCmdRev := P10_050_DI4.digitalInput_02,
    pickUpRollPosLimitFwd := P10_050_DI4.digitalInput_03,
    pickUpRollPosLimitRev := P10_050_DI4.digitalInput_04,
    babyDryerScraperOscCmd := TRUE,
    upperGroupScraperOscCmd := TRUE,
    lowerGroupScraperOscCmd := TRUE,
    paperPresenceSensor := P10_050_DI5.digitalInput_03,
    steamPressureAutoMan := paperMachineHmiCommands.dryingSectionGroup1SteamPressureAutoMan,
    steamPressureAutoSetpoint := paperMachineHmiCommands.dryingSectionGroup1SteamPressureAutoSetpoint,
    steamPressureManualSetpoint := paperMachineHmiCommands.dryingSectionGroup1SteamPressureManualSetpoint,
    steamPressureFeedback := P10_050_AI1.Channel1,
    steamPressureKp := 3,
    steamPressureTn := 8,
    steamPressureTv := 0,
    steamPressureLimLow := 0,
    steamPressureLimHigh := 60,
    upperMasterDiameter := paperMachineHmiConfig.dryingSectionGroup1UpperMasterDiameter,
    upperSlave1Diameter := paperMachineHmiConfig.dryingSectionGroup1UpperSlave1Diameter,
    lowerMasterDiameter := paperMachineHmiConfig.dryingSectionGroup1LowerMasterDiameter,
    lowerSlave1Diameter := paperMachineHmiConfig.dryingSectionGroup1LowerSlave1Diameter,
    machineConfig := paperMachineHmiConfig,
    upperMasterSpeedSetpointRPM => P13_500_UG03_1GR_UpperMaster.speedSetpoint,
    upperSlaveSpeedSetpointRPM => P13_500_UG01_1GR_UpperSlave.speedSetpoint,
    lowerMasterSpeedSetpointRPM => P13_500_UG02_1GR_LowerMaster.speedSetpoint,
    nextGroupSpeedRefMPM => dryingSectionGr1NextGroupReference,
    upperSlave1TorqueRefPct => P13_500_UG01_1GR_UpperSlave.torqueSetpoint,
    upperMasterEnable => P13_500_UG03_1GR_UpperMaster.commandWord.enableDrive,
    upperSlave1Enable => P13_500_UG01_1GR_UpperSlave.commandWord.enableDrive,
    lowerMasterEnable => P13_500_UG02_1GR_LowerMaster.commandWord.enableDrive,
    upperDryingSectionFabricStretch => P10_050_DO2.digitalOutput_10,
    upperDryingSectionFabricUnstretch => P10_050_DO2.digitalOutput_11,
    lowerDryingSectionFabricStretch => P10_050_DO2.digitalOutput_12,
    lowerDryingSectionFabricUnstretch => P10_050_DO2.digitalOutput_13,
    pickUpRollPosRunFwd => P10_050_DO2.digitalOutput_08,
    pickUpRollPosRunRev => P10_050_DO2.digitalOutput_09,
    babyDryerScraperOscRun => P10_050_DO2.digitalOutput_14,
    upperGroupScraperOscRun => P10_050_DO2.digitalOutput_15,
    lowerGroupScraperOscRun => P10_050_DO2.digitalOutput_16,
    steamPressure => paperMachineHmiStatus.dryingSectionGroup1SteamPressure,
    steamPressureControllerOutput => P10_050_AO1.Channel1,
    upperMasterSpeedMPM => paperMachineHmiStatus.dryingSectionGroup1UpperMasterSpeedMPM,
    upperSlave1SpeedMPM => paperMachineHmiStatus.dryingSectionGroup1UpperSlave1SpeedMPM,
    lowerMasterSpeedMPM => paperMachineHmiStatus.dryingSectionGroup1LowerMasterSpeedMPM,
    lowerSlave1SpeedMPM => paperMachineHmiStatus.dryingSectionGroup1LowerSlave1SpeedMPM,
    upperMasterTorque => paperMachineHmiStatus.dryingSectionGroup1UpperMasterTorque,
    upperSlave1Torque => paperMachineHmiStatus.dryingSectionGroup1UpperSlave1Torque,
    lowerMasterTorque => paperMachineHmiStatus.dryingSectionGroup1LowerMasterTorque,
    lowerSlave1Torque => paperMachineHmiStatus.dryingSectionGroup1LowerSlave1Torque); // FB_DryingSectionDriveControl_V3
END_METHOD

METHOD _501_DryingSectionGroup2DriveControl
VAR_INPUT
END_VAR
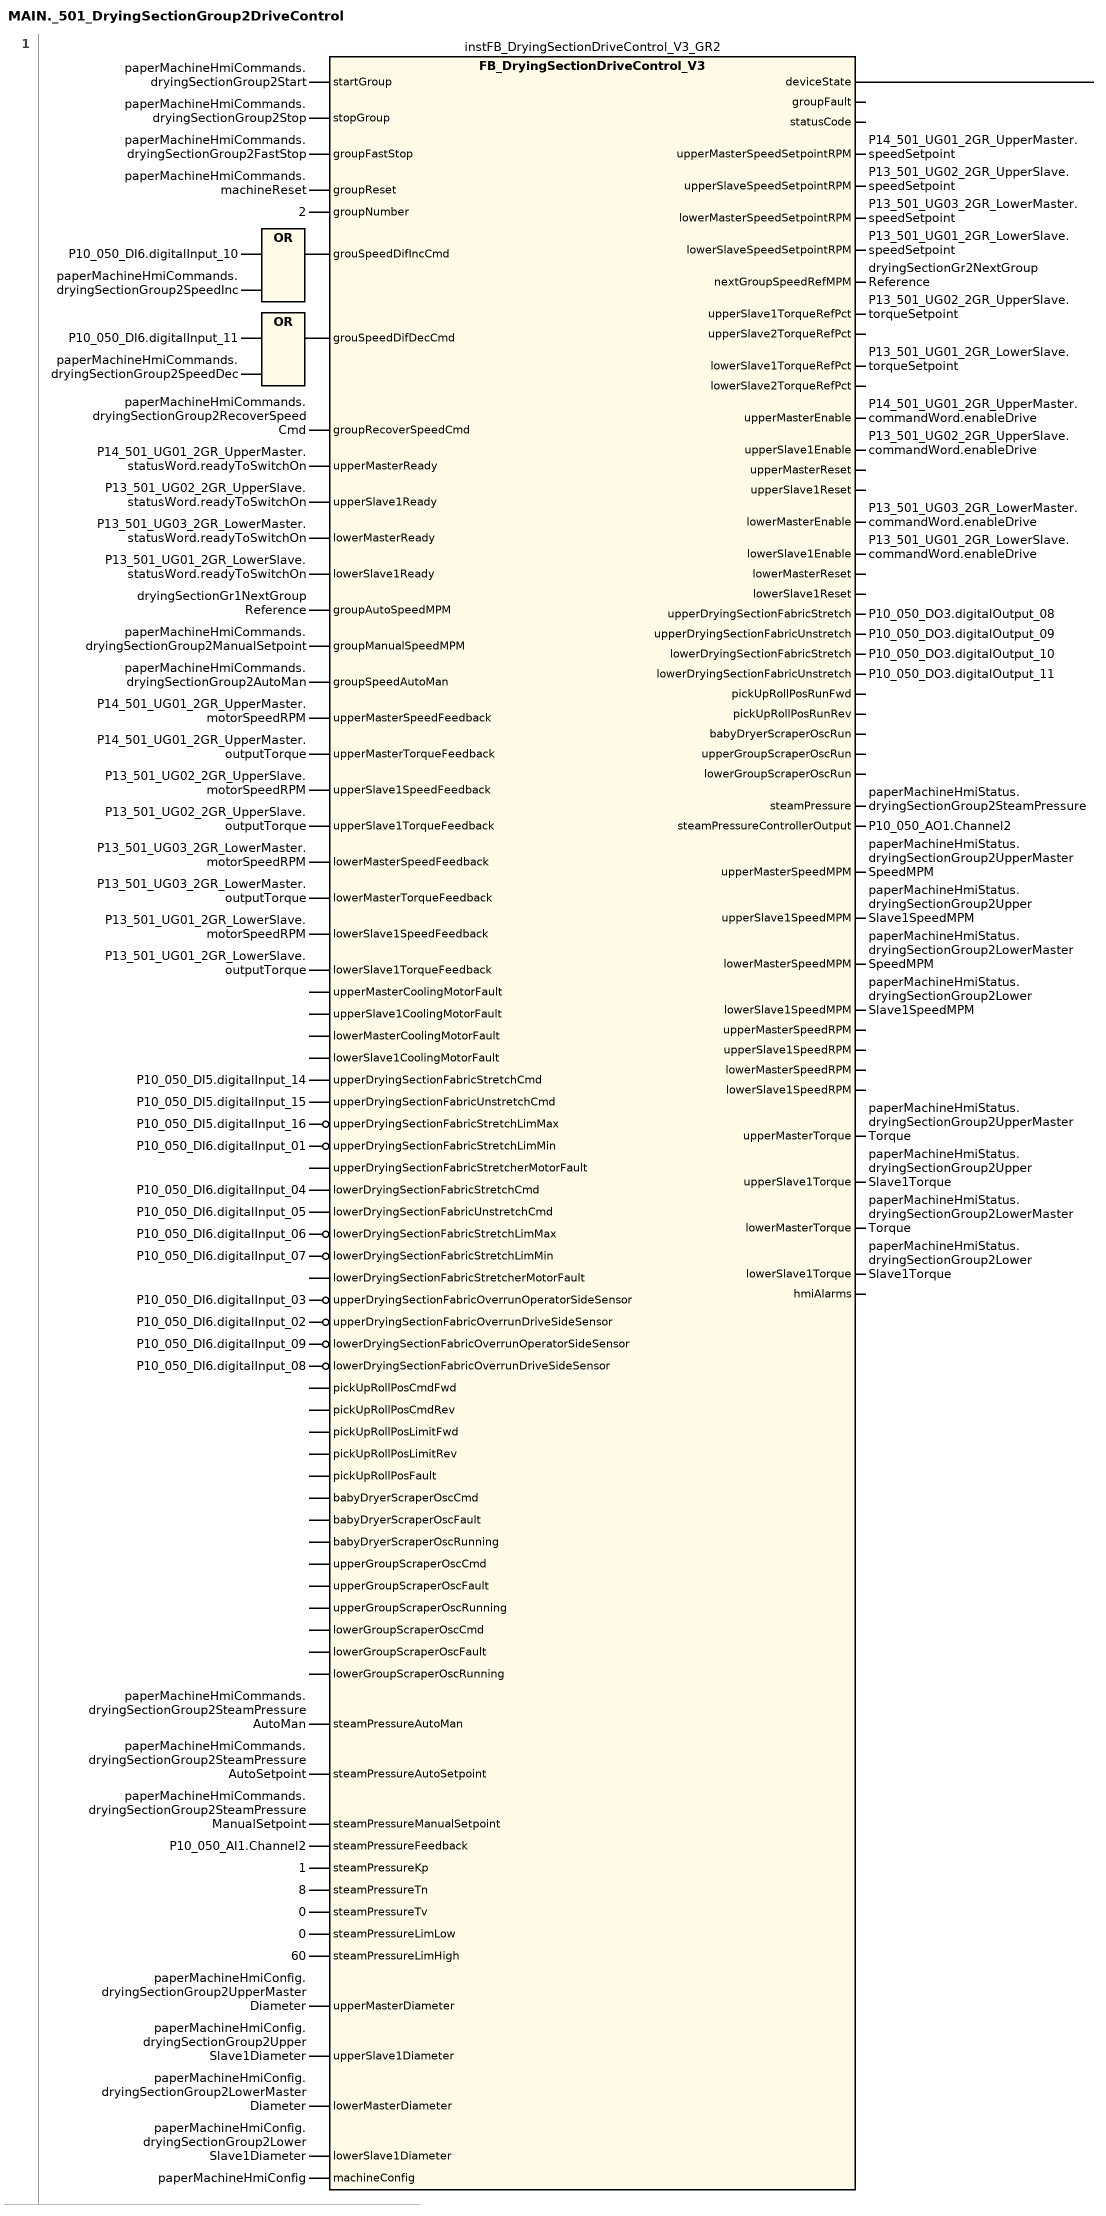
// NETWORK 1
instFB_DryingSectionDriveControl_V3_GR2(
    startGroup := paperMachineHmiCommands.dryingSectionGroup2Start,
    stopGroup := paperMachineHmiCommands.dryingSectionGroup2Stop,
    groupFastStop := paperMachineHmiCommands.dryingSectionGroup2FastStop,
    groupReset := paperMachineHmiCommands.machineReset,
    groupNumber := 2,
    grouSpeedDifIncCmd := P10_050_DI6.digitalInput_10 OR paperMachineHmiCommands.dryingSectionGroup2SpeedInc,
    grouSpeedDifDecCmd := P10_050_DI6.digitalInput_11 OR paperMachineHmiCommands.dryingSectionGroup2SpeedDec,
    groupRecoverSpeedCmd := paperMachineHmiCommands.dryingSectionGroup2RecoverSpeedCmd,
    upperMasterReady := P14_501_UG01_2GR_UpperMaster.statusWord.readyToSwitchOn,
    upperSlave1Ready := P13_501_UG02_2GR_UpperSlave.statusWord.readyToSwitchOn,
    lowerMasterReady := P13_501_UG03_2GR_LowerMaster.statusWord.readyToSwitchOn,
    lowerSlave1Ready := P13_501_UG01_2GR_LowerSlave.statusWord.readyToSwitchOn,
    groupAutoSpeedMPM := dryingSectionGr1NextGroupReference,
    groupManualSpeedMPM := paperMachineHmiCommands.dryingSectionGroup2ManualSetpoint,
    groupSpeedAutoMan := paperMachineHmiCommands.dryingSectionGroup2AutoMan,
    upperMasterSpeedFeedback := P14_501_UG01_2GR_UpperMaster.motorSpeedRPM,
    upperMasterTorqueFeedback := P14_501_UG01_2GR_UpperMaster.outputTorque,
    upperSlave1SpeedFeedback := P13_501_UG02_2GR_UpperSlave.motorSpeedRPM,
    upperSlave1TorqueFeedback := P13_501_UG02_2GR_UpperSlave.outputTorque,
    lowerMasterSpeedFeedback := P13_501_UG03_2GR_LowerMaster.motorSpeedRPM,
    lowerMasterTorqueFeedback := P13_501_UG03_2GR_LowerMaster.outputTorque,
    lowerSlave1SpeedFeedback := P13_501_UG01_2GR_LowerSlave.motorSpeedRPM,
    lowerSlave1TorqueFeedback := P13_501_UG01_2GR_LowerSlave.outputTorque,
    upperDryingSectionFabricStretchCmd := P10_050_DI5.digitalInput_14,
    upperDryingSectionFabricUnstretchCmd := P10_050_DI5.digitalInput_15,
    upperDryingSectionFabricStretchLimMax := NOT P10_050_DI5.digitalInput_16,
    upperDryingSectionFabricStretchLimMin := NOT P10_050_DI6.digitalInput_01,
    lowerDryingSectionFabricStretchCmd := P10_050_DI6.digitalInput_04,
    lowerDryingSectionFabricUnstretchCmd := P10_050_DI6.digitalInput_05,
    lowerDryingSectionFabricStretchLimMax := NOT P10_050_DI6.digitalInput_06,
    lowerDryingSectionFabricStretchLimMin := NOT P10_050_DI6.digitalInput_07,
    upperDryingSectionFabricOverrunOperatorSideSensor := NOT P10_050_DI6.digitalInput_03,
    upperDryingSectionFabricOverrunDriveSideSensor := NOT P10_050_DI6.digitalInput_02,
    lowerDryingSectionFabricOverrunOperatorSideSensor := NOT P10_050_DI6.digitalInput_09,
    lowerDryingSectionFabricOverrunDriveSideSensor := NOT P10_050_DI6.digitalInput_08,
    steamPressureAutoMan := paperMachineHmiCommands.dryingSectionGroup2SteamPressureAutoMan,
    steamPressureAutoSetpoint := paperMachineHmiCommands.dryingSectionGroup2SteamPressureAutoSetpoint,
    steamPressureManualSetpoint := paperMachineHmiCommands.dryingSectionGroup2SteamPressureManualSetpoint,
    steamPressureFeedback := P10_050_AI1.Channel2,
    steamPressureKp := 1,
    steamPressureTn := 8,
    steamPressureTv := 0,
    steamPressureLimLow := 0,
    steamPressureLimHigh := 60,
    upperMasterDiameter := paperMachineHmiConfig.dryingSectionGroup2UpperMasterDiameter,
    upperSlave1Diameter := paperMachineHmiConfig.dryingSectionGroup2UpperSlave1Diameter,
    lowerMasterDiameter := paperMachineHmiConfig.dryingSectionGroup2LowerMasterDiameter,
    lowerSlave1Diameter := paperMachineHmiConfig.dryingSectionGroup2LowerSlave1Diameter,
    machineConfig := paperMachineHmiConfig,
    upperMasterSpeedSetpointRPM => P14_501_UG01_2GR_UpperMaster.speedSetpoint,
    upperSlaveSpeedSetpointRPM => P13_501_UG02_2GR_UpperSlave.speedSetpoint,
    lowerMasterSpeedSetpointRPM => P13_501_UG03_2GR_LowerMaster.speedSetpoint,
    lowerSlaveSpeedSetpointRPM => P13_501_UG01_2GR_LowerSlave.speedSetpoint,
    nextGroupSpeedRefMPM => dryingSectionGr2NextGroupReference,
    upperSlave1TorqueRefPct => P13_501_UG02_2GR_UpperSlave.torqueSetpoint,
    lowerSlave1TorqueRefPct => P13_501_UG01_2GR_LowerSlave.torqueSetpoint,
    upperMasterEnable => P14_501_UG01_2GR_UpperMaster.commandWord.enableDrive,
    upperSlave1Enable => P13_501_UG02_2GR_UpperSlave.commandWord.enableDrive,
    lowerMasterEnable => P13_501_UG03_2GR_LowerMaster.commandWord.enableDrive,
    lowerSlave1Enable => P13_501_UG01_2GR_LowerSlave.commandWord.enableDrive,
    upperDryingSectionFabricStretch => P10_050_DO3.digitalOutput_08,
    upperDryingSectionFabricUnstretch => P10_050_DO3.digitalOutput_09,
    lowerDryingSectionFabricStretch => P10_050_DO3.digitalOutput_10,
    lowerDryingSectionFabricUnstretch => P10_050_DO3.digitalOutput_11,
    steamPressure => paperMachineHmiStatus.dryingSectionGroup2SteamPressure,
    steamPressureControllerOutput => P10_050_AO1.Channel2,
    upperMasterSpeedMPM => paperMachineHmiStatus.dryingSectionGroup2UpperMasterSpeedMPM,
    upperSlave1SpeedMPM => paperMachineHmiStatus.dryingSectionGroup2UpperSlave1SpeedMPM,
    lowerMasterSpeedMPM => paperMachineHmiStatus.dryingSectionGroup2LowerMasterSpeedMPM,
    lowerSlave1SpeedMPM => paperMachineHmiStatus.dryingSectionGroup2LowerSlave1SpeedMPM,
    upperMasterTorque => paperMachineHmiStatus.dryingSectionGroup2UpperMasterTorque,
    upperSlave1Torque => paperMachineHmiStatus.dryingSectionGroup2UpperSlave1Torque,
    lowerMasterTorque => paperMachineHmiStatus.dryingSectionGroup2LowerMasterTorque,
    lowerSlave1Torque => paperMachineHmiStatus.dryingSectionGroup2LowerSlave1Torque); // FB_DryingSectionDriveControl_V3
END_METHOD

METHOD _502_DryingSectionGroup3DriveControl
VAR_INPUT
END_VAR
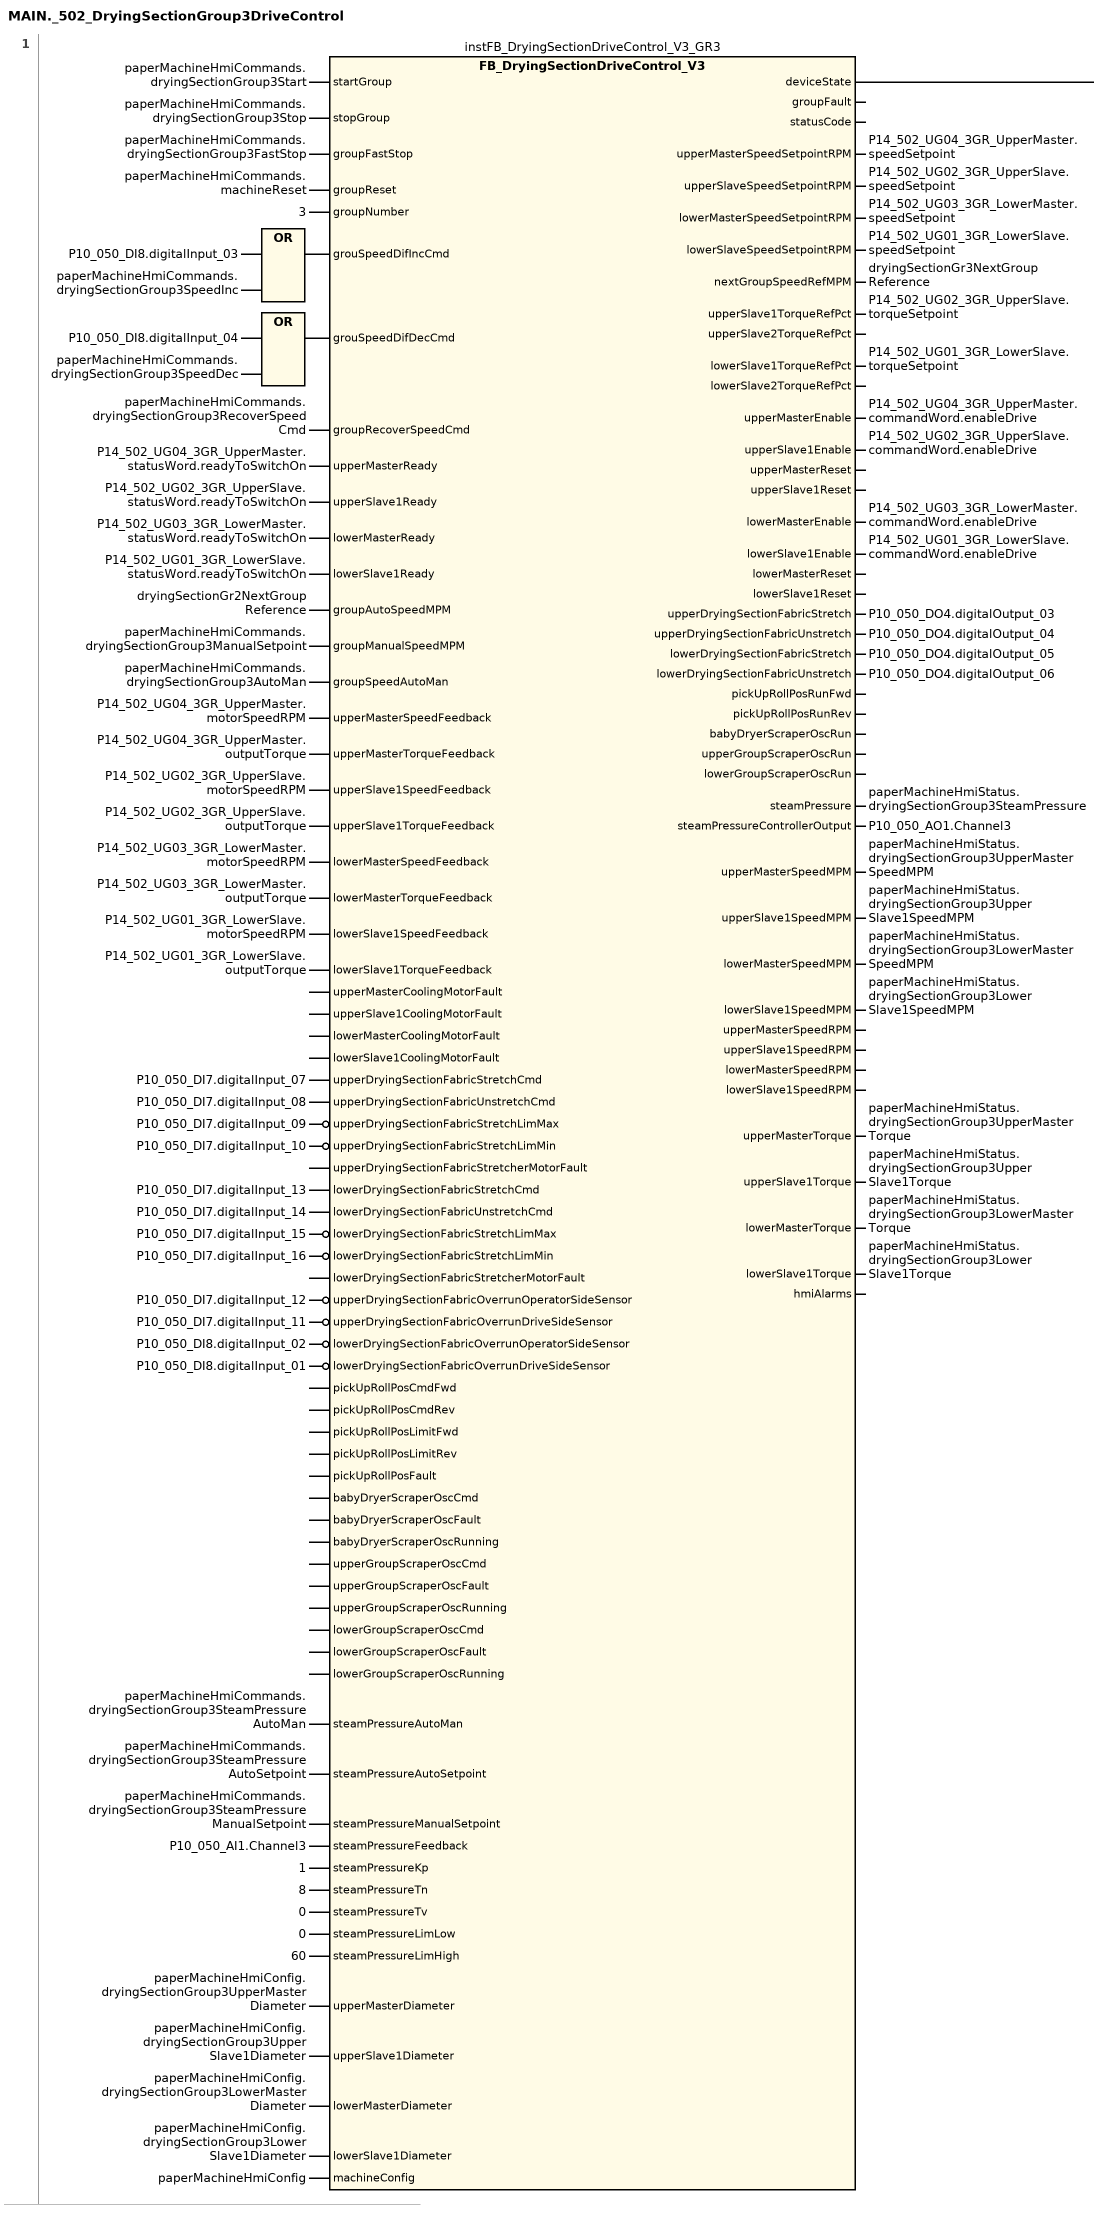
// NETWORK 1
instFB_DryingSectionDriveControl_V3_GR3(
    startGroup := paperMachineHmiCommands.dryingSectionGroup3Start,
    stopGroup := paperMachineHmiCommands.dryingSectionGroup3Stop,
    groupFastStop := paperMachineHmiCommands.dryingSectionGroup3FastStop,
    groupReset := paperMachineHmiCommands.machineReset,
    groupNumber := 3,
    grouSpeedDifIncCmd := P10_050_DI8.digitalInput_03 OR paperMachineHmiCommands.dryingSectionGroup3SpeedInc,
    grouSpeedDifDecCmd := P10_050_DI8.digitalInput_04 OR paperMachineHmiCommands.dryingSectionGroup3SpeedDec,
    groupRecoverSpeedCmd := paperMachineHmiCommands.dryingSectionGroup3RecoverSpeedCmd,
    upperMasterReady := P14_502_UG04_3GR_UpperMaster.statusWord.readyToSwitchOn,
    upperSlave1Ready := P14_502_UG02_3GR_UpperSlave.statusWord.readyToSwitchOn,
    lowerMasterReady := P14_502_UG03_3GR_LowerMaster.statusWord.readyToSwitchOn,
    lowerSlave1Ready := P14_502_UG01_3GR_LowerSlave.statusWord.readyToSwitchOn,
    groupAutoSpeedMPM := dryingSectionGr2NextGroupReference,
    groupManualSpeedMPM := paperMachineHmiCommands.dryingSectionGroup3ManualSetpoint,
    groupSpeedAutoMan := paperMachineHmiCommands.dryingSectionGroup3AutoMan,
    upperMasterSpeedFeedback := P14_502_UG04_3GR_UpperMaster.motorSpeedRPM,
    upperMasterTorqueFeedback := P14_502_UG04_3GR_UpperMaster.outputTorque,
    upperSlave1SpeedFeedback := P14_502_UG02_3GR_UpperSlave.motorSpeedRPM,
    upperSlave1TorqueFeedback := P14_502_UG02_3GR_UpperSlave.outputTorque,
    lowerMasterSpeedFeedback := P14_502_UG03_3GR_LowerMaster.motorSpeedRPM,
    lowerMasterTorqueFeedback := P14_502_UG03_3GR_LowerMaster.outputTorque,
    lowerSlave1SpeedFeedback := P14_502_UG01_3GR_LowerSlave.motorSpeedRPM,
    lowerSlave1TorqueFeedback := P14_502_UG01_3GR_LowerSlave.outputTorque,
    upperDryingSectionFabricStretchCmd := P10_050_DI7.digitalInput_07,
    upperDryingSectionFabricUnstretchCmd := P10_050_DI7.digitalInput_08,
    upperDryingSectionFabricStretchLimMax := NOT P10_050_DI7.digitalInput_09,
    upperDryingSectionFabricStretchLimMin := NOT P10_050_DI7.digitalInput_10,
    lowerDryingSectionFabricStretchCmd := P10_050_DI7.digitalInput_13,
    lowerDryingSectionFabricUnstretchCmd := P10_050_DI7.digitalInput_14,
    lowerDryingSectionFabricStretchLimMax := NOT P10_050_DI7.digitalInput_15,
    lowerDryingSectionFabricStretchLimMin := NOT P10_050_DI7.digitalInput_16,
    upperDryingSectionFabricOverrunOperatorSideSensor := NOT P10_050_DI7.digitalInput_12,
    upperDryingSectionFabricOverrunDriveSideSensor := NOT P10_050_DI7.digitalInput_11,
    lowerDryingSectionFabricOverrunOperatorSideSensor := NOT P10_050_DI8.digitalInput_02,
    lowerDryingSectionFabricOverrunDriveSideSensor := NOT P10_050_DI8.digitalInput_01,
    steamPressureAutoMan := paperMachineHmiCommands.dryingSectionGroup3SteamPressureAutoMan,
    steamPressureAutoSetpoint := paperMachineHmiCommands.dryingSectionGroup3SteamPressureAutoSetpoint,
    steamPressureManualSetpoint := paperMachineHmiCommands.dryingSectionGroup3SteamPressureManualSetpoint,
    steamPressureFeedback := P10_050_AI1.Channel3,
    steamPressureKp := 1,
    steamPressureTn := 8,
    steamPressureTv := 0,
    steamPressureLimLow := 0,
    steamPressureLimHigh := 60,
    upperMasterDiameter := paperMachineHmiConfig.dryingSectionGroup3UpperMasterDiameter,
    upperSlave1Diameter := paperMachineHmiConfig.dryingSectionGroup3UpperSlave1Diameter,
    lowerMasterDiameter := paperMachineHmiConfig.dryingSectionGroup3LowerMasterDiameter,
    lowerSlave1Diameter := paperMachineHmiConfig.dryingSectionGroup3LowerSlave1Diameter,
    machineConfig := paperMachineHmiConfig,
    upperMasterSpeedSetpointRPM => P14_502_UG04_3GR_UpperMaster.speedSetpoint,
    upperSlaveSpeedSetpointRPM => P14_502_UG02_3GR_UpperSlave.speedSetpoint,
    lowerMasterSpeedSetpointRPM => P14_502_UG03_3GR_LowerMaster.speedSetpoint,
    lowerSlaveSpeedSetpointRPM => P14_502_UG01_3GR_LowerSlave.speedSetpoint,
    nextGroupSpeedRefMPM => dryingSectionGr3NextGroupReference,
    upperSlave1TorqueRefPct => P14_502_UG02_3GR_UpperSlave.torqueSetpoint,
    lowerSlave1TorqueRefPct => P14_502_UG01_3GR_LowerSlave.torqueSetpoint,
    upperMasterEnable => P14_502_UG04_3GR_UpperMaster.commandWord.enableDrive,
    upperSlave1Enable => P14_502_UG02_3GR_UpperSlave.commandWord.enableDrive,
    lowerMasterEnable => P14_502_UG03_3GR_LowerMaster.commandWord.enableDrive,
    lowerSlave1Enable => P14_502_UG01_3GR_LowerSlave.commandWord.enableDrive,
    upperDryingSectionFabricStretch => P10_050_DO4.digitalOutput_03,
    upperDryingSectionFabricUnstretch => P10_050_DO4.digitalOutput_04,
    lowerDryingSectionFabricStretch => P10_050_DO4.digitalOutput_05,
    lowerDryingSectionFabricUnstretch => P10_050_DO4.digitalOutput_06,
    steamPressure => paperMachineHmiStatus.dryingSectionGroup3SteamPressure,
    steamPressureControllerOutput => P10_050_AO1.Channel3,
    upperMasterSpeedMPM => paperMachineHmiStatus.dryingSectionGroup3UpperMasterSpeedMPM,
    upperSlave1SpeedMPM => paperMachineHmiStatus.dryingSectionGroup3UpperSlave1SpeedMPM,
    lowerMasterSpeedMPM => paperMachineHmiStatus.dryingSectionGroup3LowerMasterSpeedMPM,
    lowerSlave1SpeedMPM => paperMachineHmiStatus.dryingSectionGroup3LowerSlave1SpeedMPM,
    upperMasterTorque => paperMachineHmiStatus.dryingSectionGroup3UpperMasterTorque,
    upperSlave1Torque => paperMachineHmiStatus.dryingSectionGroup3UpperSlave1Torque,
    lowerMasterTorque => paperMachineHmiStatus.dryingSectionGroup3LowerMasterTorque,
    lowerSlave1Torque => paperMachineHmiStatus.dryingSectionGroup3LowerSlave1Torque); // FB_DryingSectionDriveControl_V3
END_METHOD

METHOD _550_DryingSectionLubrification
VAR_INPUT
END_VAR
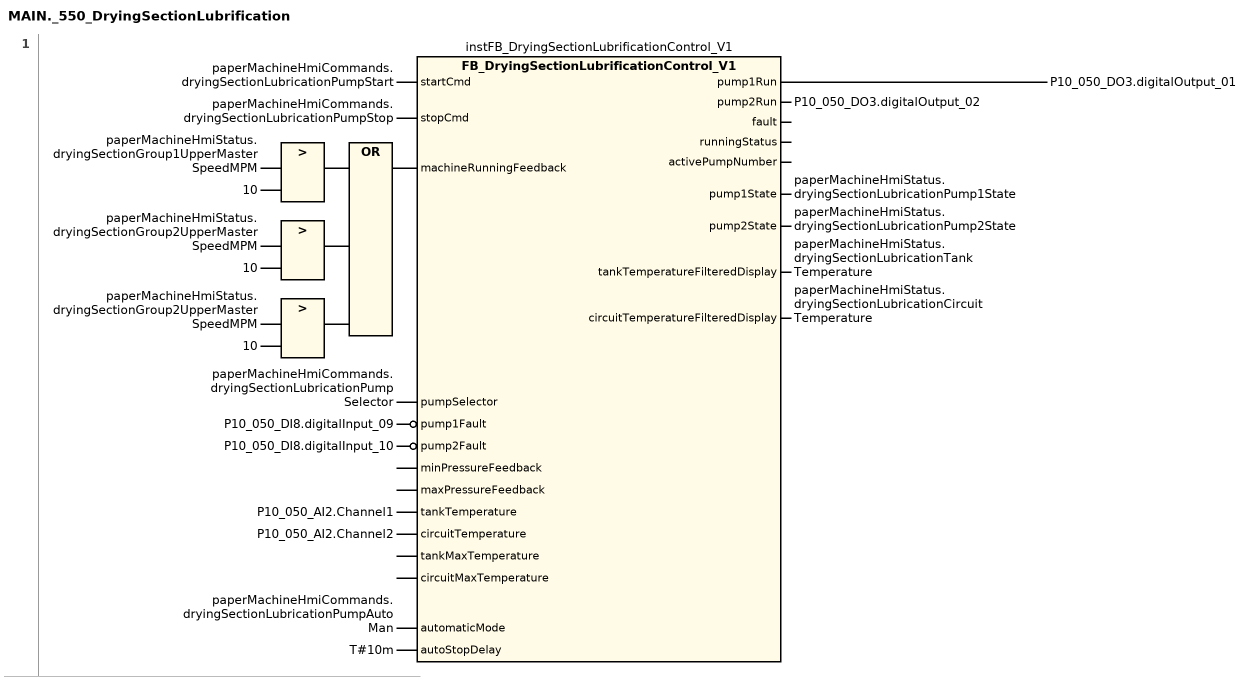
// NETWORK 1
instFB_DryingSectionLubrificationControl_V1(
    startCmd := paperMachineHmiCommands.dryingSectionLubricationPumpStart,
    stopCmd := paperMachineHmiCommands.dryingSectionLubricationPumpStop,
    machineRunningFeedback := paperMachineHmiStatus.dryingSectionGroup1UpperMasterSpeedMPM > 10 OR paperMachineHmiStatus.dryingSectionGroup2UpperMasterSpeedMPM > 10 OR paperMachineHmiStatus.dryingSectionGroup2UpperMasterSpeedMPM > 10,
    pumpSelector := paperMachineHmiCommands.dryingSectionLubricationPumpSelector,
    pump1Fault := NOT P10_050_DI8.digitalInput_09,
    pump2Fault := NOT P10_050_DI8.digitalInput_10,
    tankTemperature := P10_050_AI2.Channel1,
    circuitTemperature := P10_050_AI2.Channel2,
    automaticMode := paperMachineHmiCommands.dryingSectionLubricationPumpAutoMan,
    autoStopDelay := T#10m,
    pump2Run => P10_050_DO3.digitalOutput_02,
    pump1State => paperMachineHmiStatus.dryingSectionLubricationPump1State,
    pump2State => paperMachineHmiStatus.dryingSectionLubricationPump2State,
    tankTemperatureFilteredDisplay => paperMachineHmiStatus.dryingSectionLubricationTankTemperature,
    circuitTemperatureFilteredDisplay => paperMachineHmiStatus.dryingSectionLubricationCircuitTemperature); // FB_DryingSectionLubrificationControl_V1
P10_050_DO3.digitalOutput_01 := instFB_DryingSectionLubrificationControl_V1.pump1Run;
END_METHOD

METHOD _600_WinderGroup
VAR_INPUT
END_VAR
(*
	winderPressureSetpointOperatorSide : REAL; // EN: Controller output (operator side) / PT: Saída do controlador (lado operador)
    winderPressureSetpointDriveSide    : REAL; // EN: Controller output (drive side) / PT: Saída do controlador (lado motriz)
	winderSpeedMPM   : REAL;  // Group 2 Upper Slave 2 speed [m/min or rpm] (Velocidade do motor escravo 2 superior do grupo 2)
	winderTorque  : REAL;  // Group 2 Upper Slave 2 torque [% or Nm] (Torque do motor escravo 2 superior do grupo 2)
	winderState   : INT;   // Group 2 Upper Slave 2 state code (Estado do motor escravo 2 superior do grupo 2)
*)

(*
	// ─────────────── WINDER SECTION ───────────────
	// Start/stop and speed control commands for the winder section.
	winderSectionStart            : BOOL;  // Start Press Section (Ligar Prensa)
	winderSectionStop             : BOOL;  // Stop Press Section (Parar Prensa)
	winderSectionAutoMan          : BOOL;  // 1 = Auto / 0 = Manual mode (Modo automático/manual)
	winderSectionManualSetpoint   : REAL;  // Manual speed setpoint [m/min] (Setpoint manual)
	winderSectionSpeedInc         : BOOL;  // Increase speed manually (Aumentar velocidade)
	winderSectionSpeedDec         : BOOL;  // Decrease speed manually (Diminuir velocidade)
	winderSectionRecoverSpeedCmd  : BOOL;  // Temporarily recover speed (Recuperar velocidade)
	winderSectionRecoverIncrement : REAL;  // Recovery speed increment [m/min or %] (Incremento de recuperação)


  // Pressure fine adjustments for rider roll
    winderPressureOperatorSideIncCmd : BOOL; // EN: Increase operator-side pressure / PT: Aumenta a pressão no lado do operador
    winderPressureOperatorSideDecCmd : BOOL; // EN: Decrease operator-side pressure / PT: Diminui a pressão no lado do operador

    winderPressureDriveSideIncCmd    : BOOL; // EN: Increase drive-side pressure / PT: Aumenta a pressão no lado motriz
    winderPressureDriveSideDecCmd    : BOOL; // EN: Decrease drive-side pressure / PT: Diminui a pressão no lado motriz

	winderRiderRollWorkPositionCmd	: BOOL;
	winderRiderRollReleasePositionCmd	: BOOL;
	
    //==============================================================
    // CORE LOCK (CHUCK LOCKING SYSTEM)
    //==============================================================
    winderCoreLockAutoMan         : BOOL;  // EN: Core lock mode (0=Manual, 1=Auto) / PT: Modo do travamento do mandril (0=Manual, 1=Automático)
    winderCoreLockCmd             : BOOL;  // EN: Lock core chucks / PT: Travar mandril (core chucks)
    winderCoreUnlockCmd           : BOOL;  // EN: Unlock core chucks / PT: Destravar mandril

	//==============================================================
    // CORE LOCK (CHUCK LOCKING SYSTEM)
    //==============================================================
	winderCoreAceleratorEngageCmd : BOOL;
	winderCoreAceleratorDisengageCmd : BOOL;
	
    //==============================================================
    // CORE BRAKE CONTROL
    //==============================================================
    winderCoreBrakeAutoMan        : BOOL;  // EN: Core brake mode (0=Manual, 1=Auto) / PT: Modo de freio do mandril (0=Manual, 1=Automático)
    winderCoreBrakeEnableCmd      : BOOL;  // EN: Enable core brake / PT: Habilita o freio do mandril
    winderCoreBrakeDisableCmd     : BOOL;  // EN: Disable core brake / PT: Desabilita o freio do mandril	
	
	// ─────────────── WINDER SECTION ───────────────
	// Start/stop and speed control commands for the winder section.
	winderSectionStart            : BOOL;  // Start Press Section (Ligar Prensa)
	winderSectionStop             : BOOL;  // Stop Press Section (Parar Prensa)
	winderSectionAutoMan          : BOOL;  // 1 = Auto / 0 = Manual mode (Modo automático/manual)
	winderSectionManualSetpoint   : REAL;  // Manual speed setpoint [m/min] (Setpoint manual)
	winderSectionSpeedInc         : BOOL;  // Increase speed manually (Aumentar velocidade)
	winderSectionSpeedDec         : BOOL;  // Decrease speed manually (Diminuir velocidade)
	winderSectionRecoverSpeedCmd  : BOOL;  // Temporarily recover speed (Recuperar velocidade)
	winderSectionRecoverIncrement : REAL;  // Recovery speed increment [m/min or %] (Incremento de recuperação)
	
    //==============================================================
    // CORE BRAKE CONTROL
    //==============================================================
    winderCoreBrakeAutoMan        : BOOL;  // EN: Core brake mode (0=Manual, 1=Auto) / PT: Modo de freio do mandril (0=Manual, 1=Automático)
    winderCoreBrakeEnableCmd      : BOOL;  // EN: Enable core brake / PT: Habilita o freio do mandril
    winderCoreBrakeDisableCmd     : BOOL;  // EN: Disable core brake / PT: Desabilita o freio do mandril	
	
	winderCorePositioningArmFwdCmd      : BOOL;  // EN: Command to move arm forward / PT: Comando para avançar o braço posicionador
    winderCorePositioningArmRevCmd      : BOOL;  // EN: Command to move arm backward / PT: Comando para recuar o braço posicionador

    winderCorePositioningArmPosLimitFwd : BOOL;  // EN: Forward limit switch / PT: Fim de curso avançado
    winderCorePositioningArmPosLimitRev : BOOL;  // EN: Reverse limit switch / PT: Fim de curso recuado	
*)
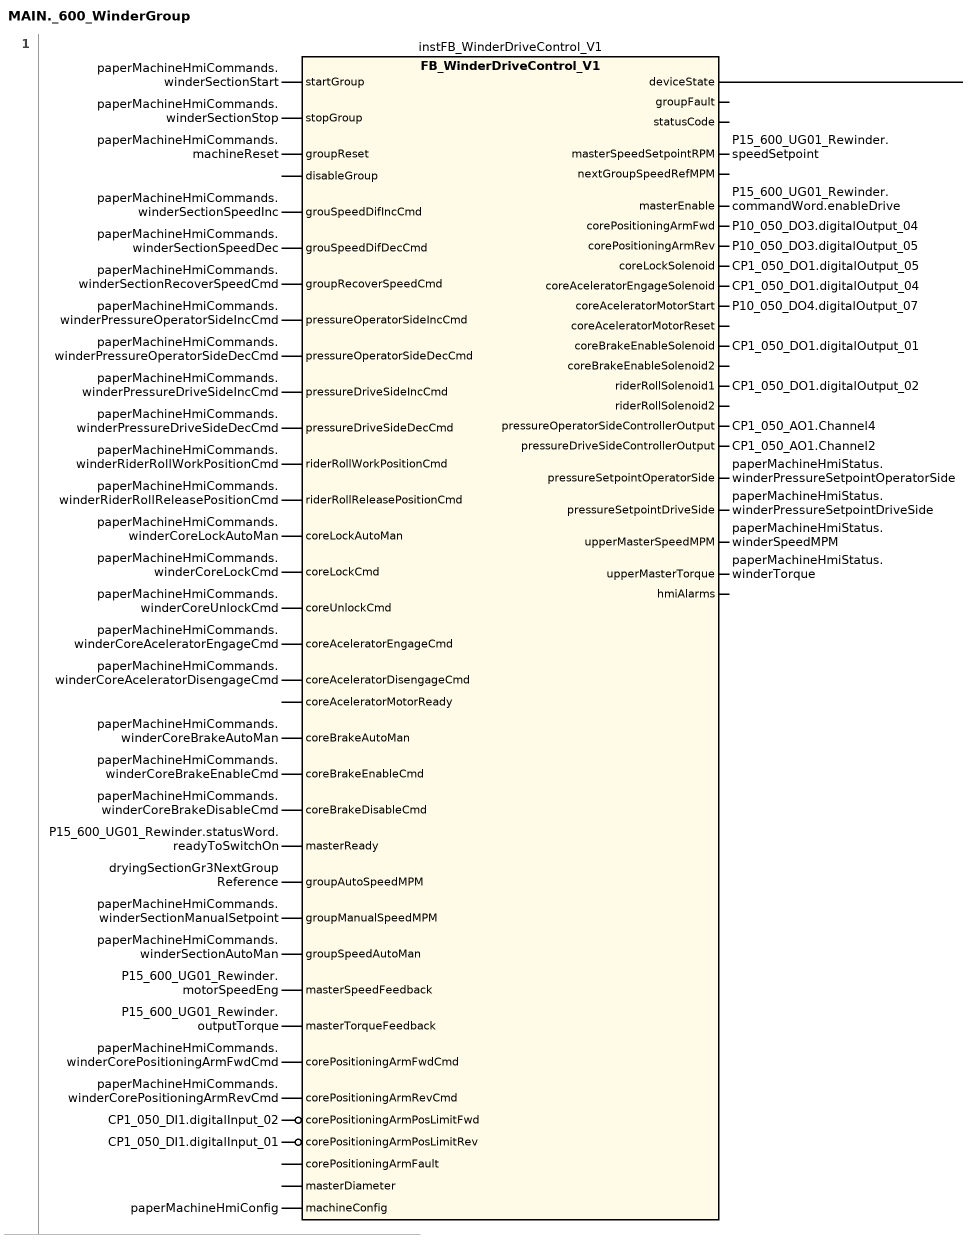
// NETWORK 1
instFB_WinderDriveControl_V1(
    startGroup := paperMachineHmiCommands.winderSectionStart,
    stopGroup := paperMachineHmiCommands.winderSectionStop,
    groupReset := paperMachineHmiCommands.machineReset,
    grouSpeedDifIncCmd := paperMachineHmiCommands.winderSectionSpeedInc,
    grouSpeedDifDecCmd := paperMachineHmiCommands.winderSectionSpeedDec,
    groupRecoverSpeedCmd := paperMachineHmiCommands.winderSectionRecoverSpeedCmd,
    pressureOperatorSideIncCmd := paperMachineHmiCommands.winderPressureOperatorSideIncCmd,
    pressureOperatorSideDecCmd := paperMachineHmiCommands.winderPressureOperatorSideDecCmd,
    pressureDriveSideIncCmd := paperMachineHmiCommands.winderPressureDriveSideIncCmd,
    pressureDriveSideDecCmd := paperMachineHmiCommands.winderPressureDriveSideDecCmd,
    riderRollWorkPositionCmd := paperMachineHmiCommands.winderRiderRollWorkPositionCmd,
    riderRollReleasePositionCmd := paperMachineHmiCommands.winderRiderRollReleasePositionCmd,
    coreLockAutoMan := paperMachineHmiCommands.winderCoreLockAutoMan,
    coreLockCmd := paperMachineHmiCommands.winderCoreLockCmd,
    coreUnlockCmd := paperMachineHmiCommands.winderCoreUnlockCmd,
    coreAceleratorEngageCmd := paperMachineHmiCommands.winderCoreAceleratorEngageCmd,
    coreAceleratorDisengageCmd := paperMachineHmiCommands.winderCoreAceleratorDisengageCmd,
    coreBrakeAutoMan := paperMachineHmiCommands.winderCoreBrakeAutoMan,
    coreBrakeEnableCmd := paperMachineHmiCommands.winderCoreBrakeEnableCmd,
    coreBrakeDisableCmd := paperMachineHmiCommands.winderCoreBrakeDisableCmd,
    masterReady := P15_600_UG01_Rewinder.statusWord.readyToSwitchOn,
    groupAutoSpeedMPM := dryingSectionGr3NextGroupReference,
    groupManualSpeedMPM := paperMachineHmiCommands.winderSectionManualSetpoint,
    groupSpeedAutoMan := paperMachineHmiCommands.winderSectionAutoMan,
    masterSpeedFeedback := P15_600_UG01_Rewinder.motorSpeedEng,
    masterTorqueFeedback := P15_600_UG01_Rewinder.outputTorque,
    corePositioningArmFwdCmd := paperMachineHmiCommands.winderCorePositioningArmFwdCmd,
    corePositioningArmRevCmd := paperMachineHmiCommands.winderCorePositioningArmRevCmd,
    corePositioningArmPosLimitFwd := NOT CP1_050_DI1.digitalInput_02,
    corePositioningArmPosLimitRev := NOT CP1_050_DI1.digitalInput_01,
    machineConfig := paperMachineHmiConfig,
    masterSpeedSetpointRPM => P15_600_UG01_Rewinder.speedSetpoint,
    masterEnable => P15_600_UG01_Rewinder.commandWord.enableDrive,
    corePositioningArmFwd => P10_050_DO3.digitalOutput_04,
    corePositioningArmRev => P10_050_DO3.digitalOutput_05,
    coreLockSolenoid => CP1_050_DO1.digitalOutput_05,
    coreAceleratorEngageSolenoid => CP1_050_DO1.digitalOutput_04,
    coreAceleratorMotorStart => P10_050_DO4.digitalOutput_07,
    coreBrakeEnableSolenoid => CP1_050_DO1.digitalOutput_01,
    riderRollSolenoid1 => CP1_050_DO1.digitalOutput_02,
    pressureOperatorSideControllerOutput => CP1_050_AO1.Channel4,
    pressureDriveSideControllerOutput => CP1_050_AO1.Channel2,
    pressureSetpointOperatorSide => paperMachineHmiStatus.winderPressureSetpointOperatorSide,
    pressureSetpointDriveSide => paperMachineHmiStatus.winderPressureSetpointDriveSide,
    upperMasterSpeedMPM => paperMachineHmiStatus.winderSpeedMPM,
    upperMasterTorque => paperMachineHmiStatus.winderTorque); // FB_WinderDriveControl_V1
END_METHOD

METHOD _888_Alarms
VAR_INPUT
END_VAR
(*

FB_AlarmControl
*)
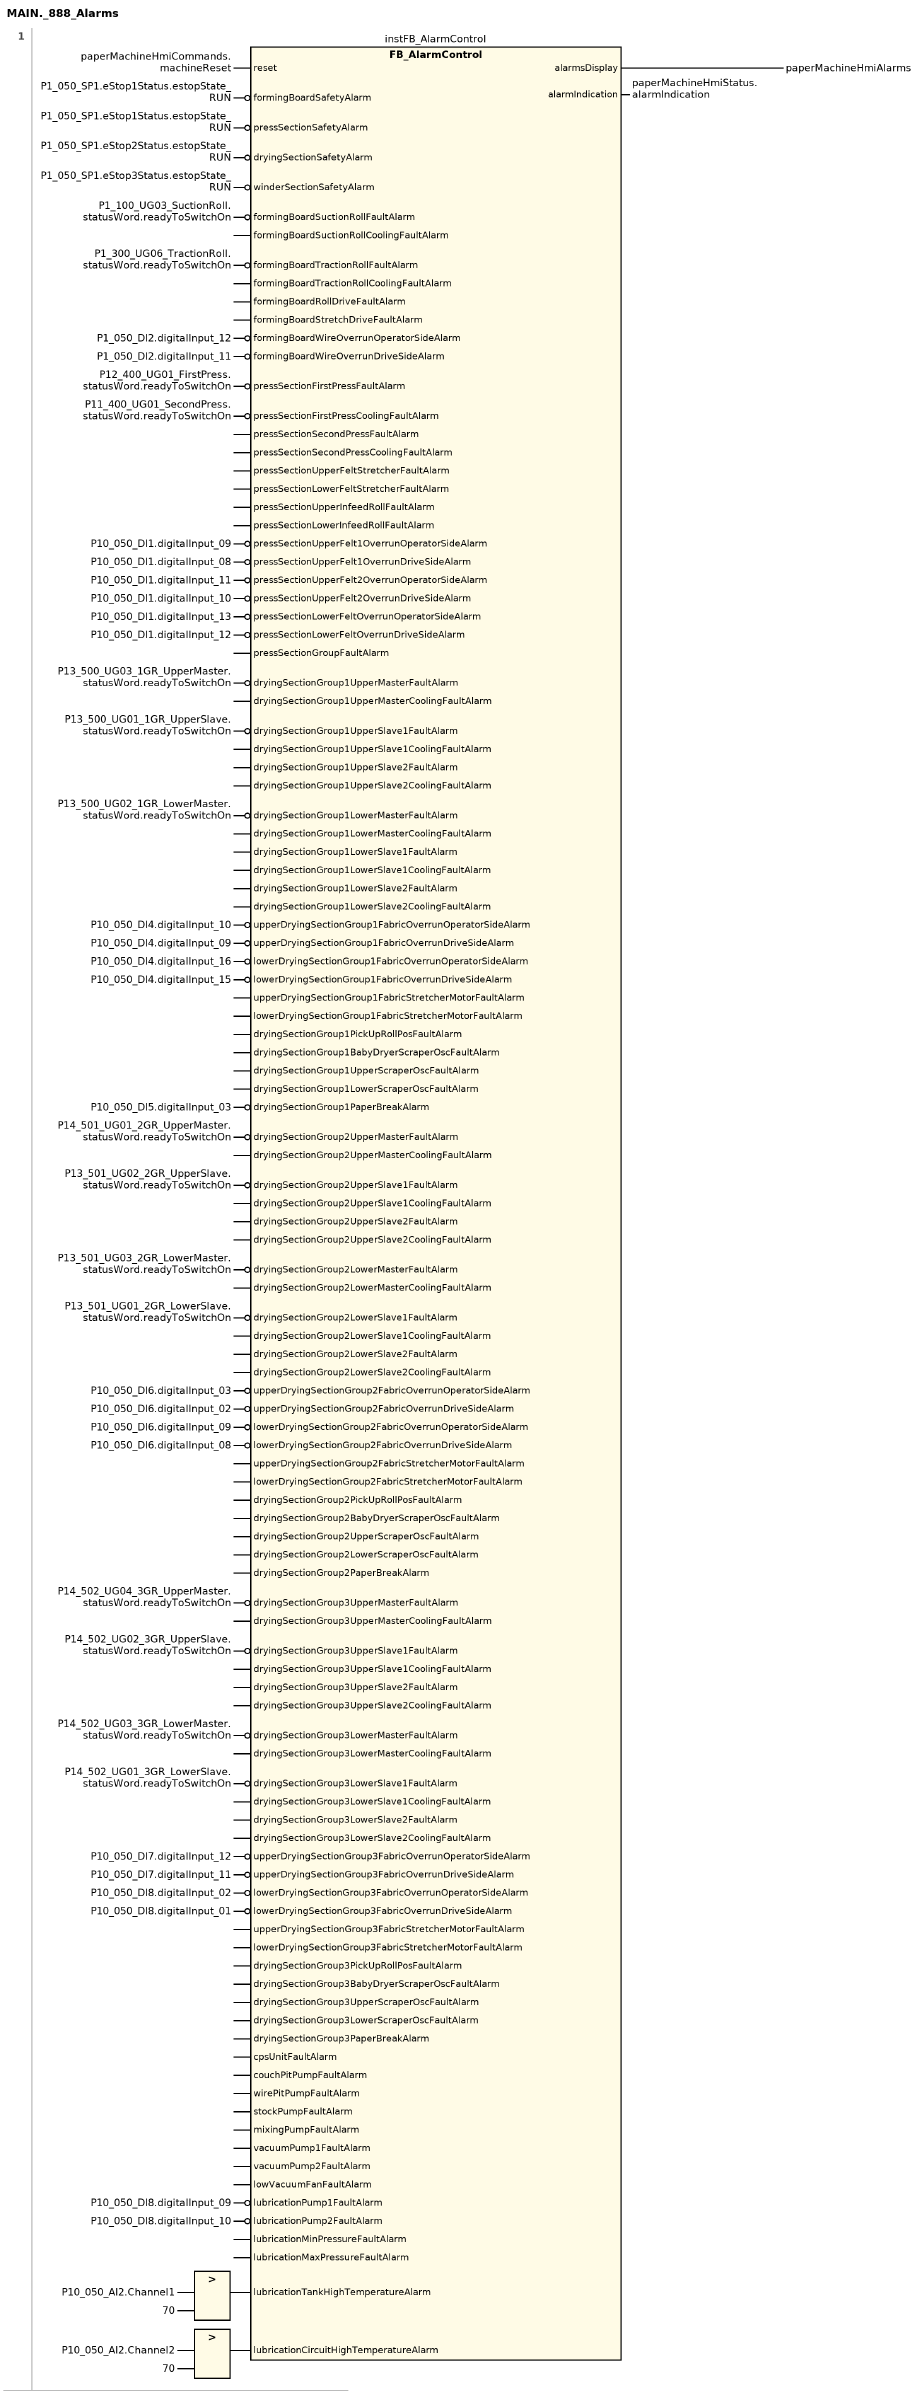
// NETWORK 1
instFB_AlarmControl(
    reset := paperMachineHmiCommands.machineReset,
    formingBoardSafetyAlarm := NOT P1_050_SP1.eStop1Status.estopState_RUN,
    pressSectionSafetyAlarm := NOT P1_050_SP1.eStop1Status.estopState_RUN,
    dryingSectionSafetyAlarm := NOT P1_050_SP1.eStop2Status.estopState_RUN,
    winderSectionSafetyAlarm := NOT P1_050_SP1.eStop3Status.estopState_RUN,
    formingBoardSuctionRollFaultAlarm := NOT P1_100_UG03_SuctionRoll.statusWord.readyToSwitchOn,
    formingBoardTractionRollFaultAlarm := NOT P1_300_UG06_TractionRoll.statusWord.readyToSwitchOn,
    formingBoardWireOverrunOperatorSideAlarm := NOT P1_050_DI2.digitalInput_12,
    formingBoardWireOverrunDriveSideAlarm := NOT P1_050_DI2.digitalInput_11,
    pressSectionFirstPressFaultAlarm := NOT P12_400_UG01_FirstPress.statusWord.readyToSwitchOn,
    pressSectionFirstPressCoolingFaultAlarm := NOT P11_400_UG01_SecondPress.statusWord.readyToSwitchOn,
    pressSectionUpperFelt1OverrunOperatorSideAlarm := NOT P10_050_DI1.digitalInput_09,
    pressSectionUpperFelt1OverrunDriveSideAlarm := NOT P10_050_DI1.digitalInput_08,
    pressSectionUpperFelt2OverrunOperatorSideAlarm := NOT P10_050_DI1.digitalInput_11,
    pressSectionUpperFelt2OverrunDriveSideAlarm := NOT P10_050_DI1.digitalInput_10,
    pressSectionLowerFeltOverrunOperatorSideAlarm := NOT P10_050_DI1.digitalInput_13,
    pressSectionLowerFeltOverrunDriveSideAlarm := NOT P10_050_DI1.digitalInput_12,
    dryingSectionGroup1UpperMasterFaultAlarm := NOT P13_500_UG03_1GR_UpperMaster.statusWord.readyToSwitchOn,
    dryingSectionGroup1UpperSlave1FaultAlarm := NOT P13_500_UG01_1GR_UpperSlave.statusWord.readyToSwitchOn,
    dryingSectionGroup1LowerMasterFaultAlarm := NOT P13_500_UG02_1GR_LowerMaster.statusWord.readyToSwitchOn,
    upperDryingSectionGroup1FabricOverrunOperatorSideAlarm := NOT P10_050_DI4.digitalInput_10,
    upperDryingSectionGroup1FabricOverrunDriveSideAlarm := NOT P10_050_DI4.digitalInput_09,
    lowerDryingSectionGroup1FabricOverrunOperatorSideAlarm := NOT P10_050_DI4.digitalInput_16,
    lowerDryingSectionGroup1FabricOverrunDriveSideAlarm := NOT P10_050_DI4.digitalInput_15,
    dryingSectionGroup1PaperBreakAlarm := NOT P10_050_DI5.digitalInput_03,
    dryingSectionGroup2UpperMasterFaultAlarm := NOT P14_501_UG01_2GR_UpperMaster.statusWord.readyToSwitchOn,
    dryingSectionGroup2UpperSlave1FaultAlarm := NOT P13_501_UG02_2GR_UpperSlave.statusWord.readyToSwitchOn,
    dryingSectionGroup2LowerMasterFaultAlarm := NOT P13_501_UG03_2GR_LowerMaster.statusWord.readyToSwitchOn,
    dryingSectionGroup2LowerSlave1FaultAlarm := NOT P13_501_UG01_2GR_LowerSlave.statusWord.readyToSwitchOn,
    upperDryingSectionGroup2FabricOverrunOperatorSideAlarm := NOT P10_050_DI6.digitalInput_03,
    upperDryingSectionGroup2FabricOverrunDriveSideAlarm := NOT P10_050_DI6.digitalInput_02,
    lowerDryingSectionGroup2FabricOverrunOperatorSideAlarm := NOT P10_050_DI6.digitalInput_09,
    lowerDryingSectionGroup2FabricOverrunDriveSideAlarm := NOT P10_050_DI6.digitalInput_08,
    dryingSectionGroup3UpperMasterFaultAlarm := NOT P14_502_UG04_3GR_UpperMaster.statusWord.readyToSwitchOn,
    dryingSectionGroup3UpperSlave1FaultAlarm := NOT P14_502_UG02_3GR_UpperSlave.statusWord.readyToSwitchOn,
    dryingSectionGroup3LowerMasterFaultAlarm := NOT P14_502_UG03_3GR_LowerMaster.statusWord.readyToSwitchOn,
    dryingSectionGroup3LowerSlave1FaultAlarm := NOT P14_502_UG01_3GR_LowerSlave.statusWord.readyToSwitchOn,
    upperDryingSectionGroup3FabricOverrunOperatorSideAlarm := NOT P10_050_DI7.digitalInput_12,
    upperDryingSectionGroup3FabricOverrunDriveSideAlarm := NOT P10_050_DI7.digitalInput_11,
    lowerDryingSectionGroup3FabricOverrunOperatorSideAlarm := NOT P10_050_DI8.digitalInput_02,
    lowerDryingSectionGroup3FabricOverrunDriveSideAlarm := NOT P10_050_DI8.digitalInput_01,
    lubricationPump1FaultAlarm := NOT P10_050_DI8.digitalInput_09,
    lubricationPump2FaultAlarm := NOT P10_050_DI8.digitalInput_10,
    lubricationTankHighTemperatureAlarm := P10_050_AI2.Channel1 > 70,
    lubricationCircuitHighTemperatureAlarm := P10_050_AI2.Channel2 > 70,
    alarmIndication => paperMachineHmiStatus.alarmIndication); // FB_AlarmControl
paperMachineHmiAlarms := instFB_AlarmControl.alarmsDisplay;
END_METHOD

METHOD _CentrifugalPressureScreenControl
VAR_INPUT
END_VAR
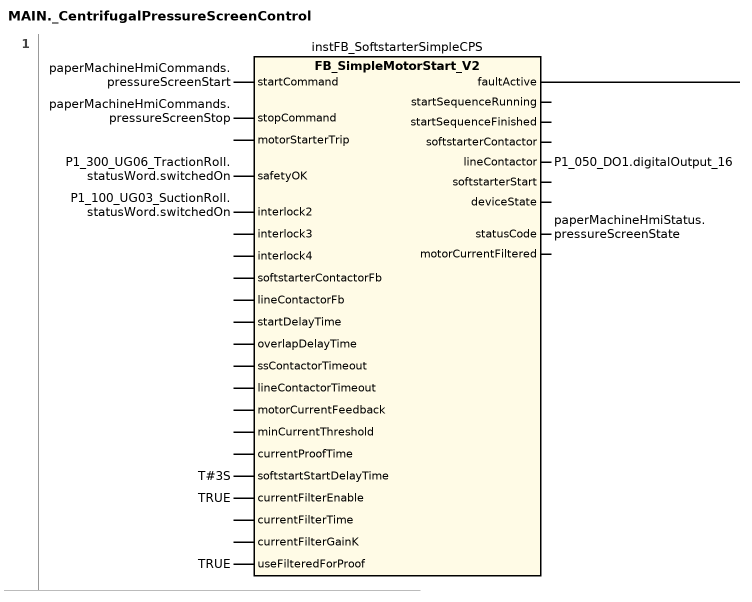
// NETWORK 1
instFB_SoftstarterSimpleCPS(
    startCommand := paperMachineHmiCommands.pressureScreenStart,
    stopCommand := paperMachineHmiCommands.pressureScreenStop,
    safetyOK := P1_300_UG06_TractionRoll.statusWord.switchedOn,
    interlock2 := P1_100_UG03_SuctionRoll.statusWord.switchedOn,
    softstartStartDelayTime := T#3S,
    currentFilterEnable := TRUE,
    useFilteredForProof := TRUE,
    lineContactor => P1_050_DO1.digitalOutput_16,
    statusCode => paperMachineHmiStatus.pressureScreenState); // FB_SimpleMotorStart_V2
END_METHOD

METHOD _CouchPitMixerControl
VAR_INPUT
END_VAR
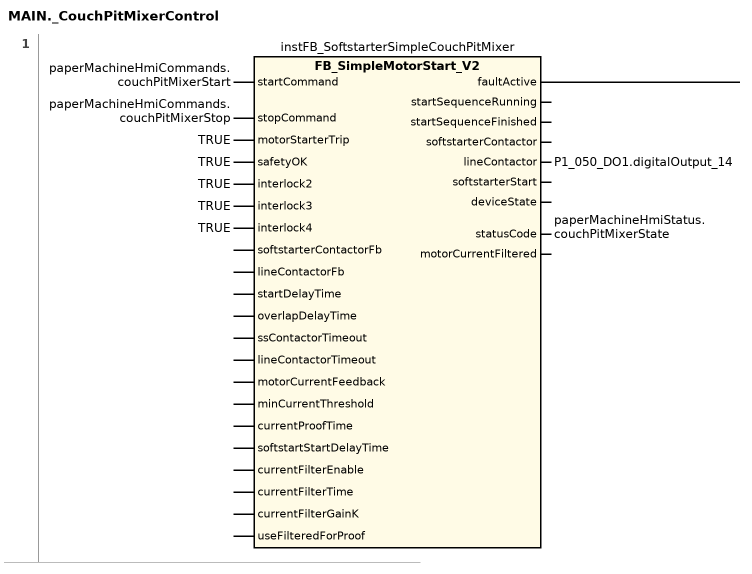
// NETWORK 1
instFB_SoftstarterSimpleCouchPitMixer(
    startCommand := paperMachineHmiCommands.couchPitMixerStart,
    stopCommand := paperMachineHmiCommands.couchPitMixerStop,
    motorStarterTrip := TRUE,
    safetyOK := TRUE,
    interlock2 := TRUE,
    interlock3 := TRUE,
    interlock4 := TRUE,
    lineContactor => P1_050_DO1.digitalOutput_14,
    statusCode => paperMachineHmiStatus.couchPitMixerState); // FB_SimpleMotorStart_V2
END_METHOD

METHOD _CouchPitPumpControl
VAR_INPUT
END_VAR
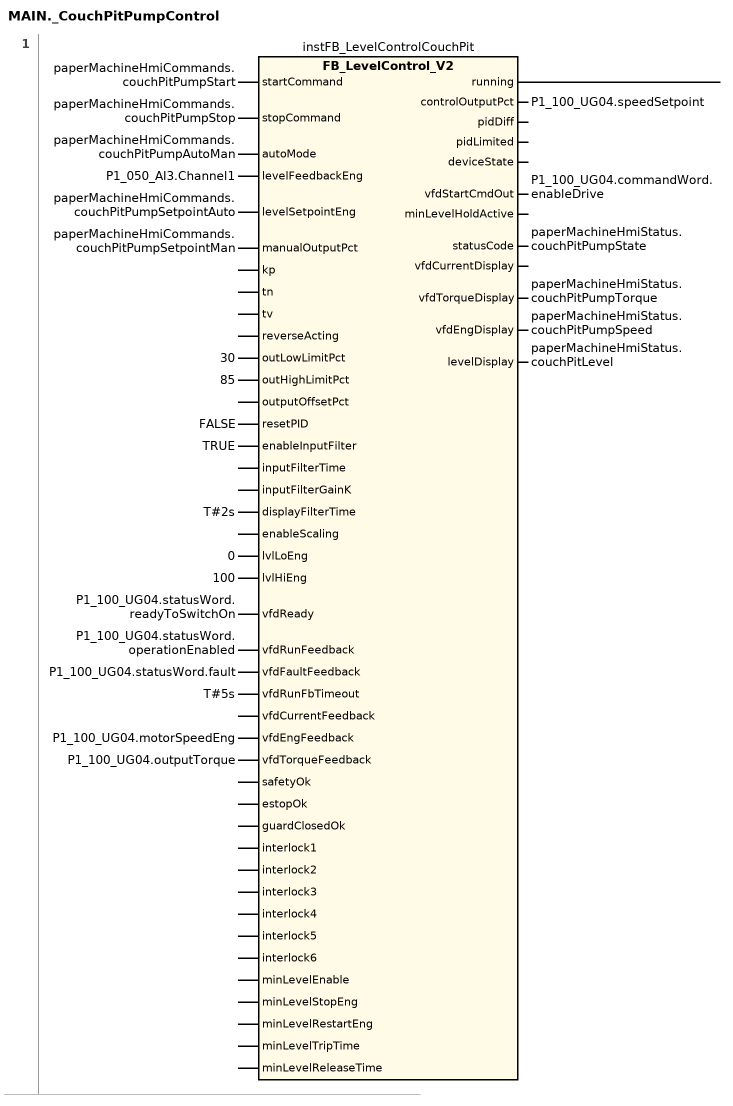
// NETWORK 1
instFB_LevelControlCouchPit(
    startCommand := paperMachineHmiCommands.couchPitPumpStart,
    stopCommand := paperMachineHmiCommands.couchPitPumpStop,
    autoMode := paperMachineHmiCommands.couchPitPumpAutoMan,
    levelFeedbackEng := P1_050_AI3.Channel1,
    levelSetpointEng := paperMachineHmiCommands.couchPitPumpSetpointAuto,
    manualOutputPct := paperMachineHmiCommands.couchPitPumpSetpointMan,
    outLowLimitPct := 30,
    outHighLimitPct := 85,
    resetPID := FALSE,
    enableInputFilter := TRUE,
    displayFilterTime := T#2s,
    lvlLoEng := 0,
    lvlHiEng := 100,
    vfdReady := P1_100_UG04.statusWord.readyToSwitchOn,
    vfdRunFeedback := P1_100_UG04.statusWord.operationEnabled,
    vfdFaultFeedback := P1_100_UG04.statusWord.fault,
    vfdRunFbTimeout := T#5s,
    vfdEngFeedback := P1_100_UG04.motorSpeedEng,
    vfdTorqueFeedback := P1_100_UG04.outputTorque,
    controlOutputPct => P1_100_UG04.speedSetpoint,
    vfdStartCmdOut => P1_100_UG04.commandWord.enableDrive,
    statusCode => paperMachineHmiStatus.couchPitPumpState,
    vfdTorqueDisplay => paperMachineHmiStatus.couchPitPumpTorque,
    vfdEngDisplay => paperMachineHmiStatus.couchPitPumpSpeed,
    levelDisplay => paperMachineHmiStatus.couchPitLevel); // FB_LevelControl_V2
END_METHOD

METHOD _FunctionBlockTest
VAR_INPUT
END_VAR
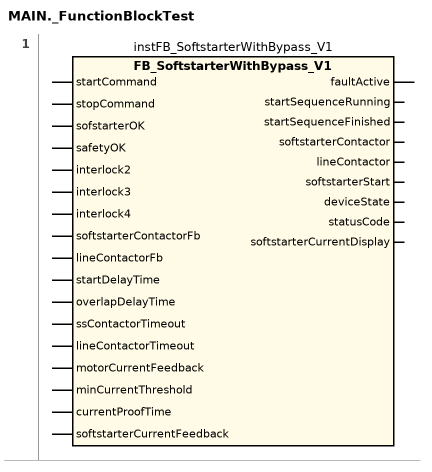
// NETWORK 1
instFB_SoftstarterWithBypass_V1(); // FB_SoftstarterWithBypass_V1
END_METHOD

METHOD _HeadBoxAuxiliaryControls
VAR_INPUT
END_VAR
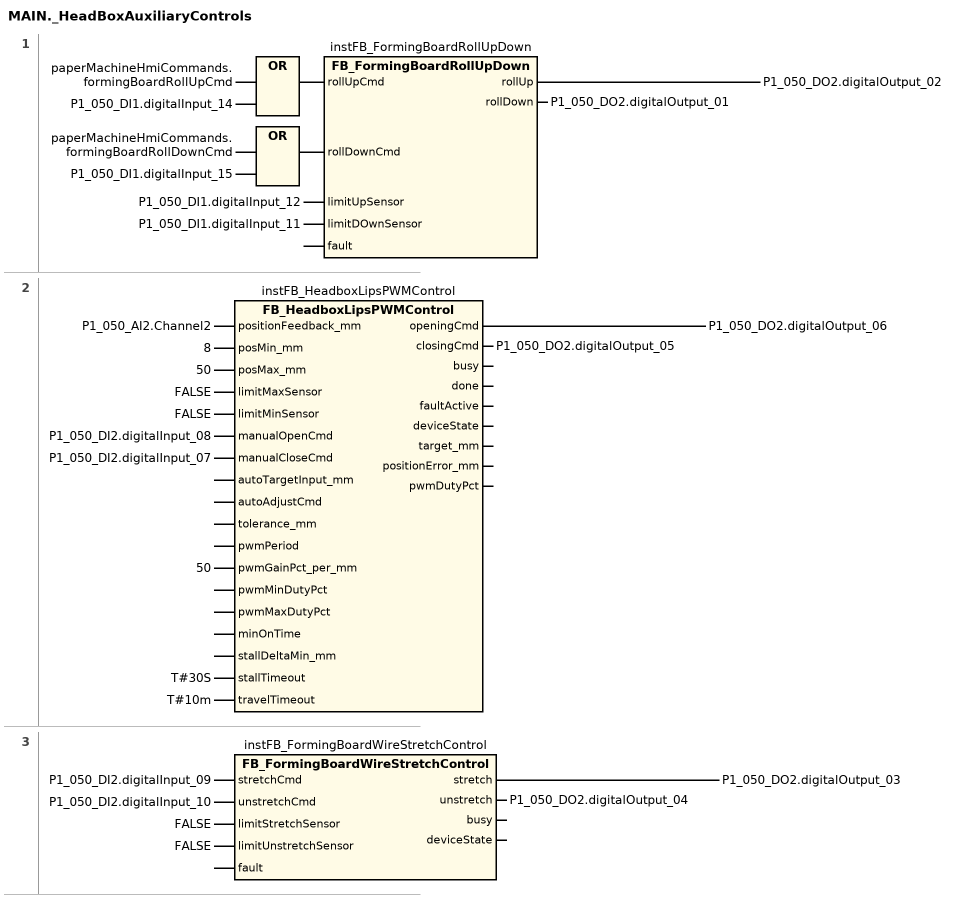
// NETWORK 1
instFB_FormingBoardRollUpDown(
    rollUpCmd := paperMachineHmiCommands.formingBoardRollUpCmd OR P1_050_DI1.digitalInput_14,
    rollDownCmd := paperMachineHmiCommands.formingBoardRollDownCmd OR P1_050_DI1.digitalInput_15,
    limitUpSensor := P1_050_DI1.digitalInput_12,
    limitDOwnSensor := P1_050_DI1.digitalInput_11,
    rollDown => P1_050_DO2.digitalOutput_01); // FB_FormingBoardRollUpDown
P1_050_DO2.digitalOutput_02 := instFB_FormingBoardRollUpDown.rollUp;

// NETWORK 2
instFB_HeadboxLipsPWMControl(
    positionFeedback_mm := P1_050_AI2.Channel2,
    posMin_mm := 8,
    posMax_mm := 50,
    limitMaxSensor := FALSE,
    limitMinSensor := FALSE,
    manualOpenCmd := P1_050_DI2.digitalInput_08,
    manualCloseCmd := P1_050_DI2.digitalInput_07,
    pwmGainPct_per_mm := 50,
    stallTimeout := T#30S,
    travelTimeout := T#10m,
    closingCmd => P1_050_DO2.digitalOutput_05); // FB_HeadboxLipsPWMControl
P1_050_DO2.digitalOutput_06 := instFB_HeadboxLipsPWMControl.openingCmd;

// NETWORK 3
instFB_FormingBoardWireStretchControl(
    stretchCmd := P1_050_DI2.digitalInput_09,
    unstretchCmd := P1_050_DI2.digitalInput_10,
    limitStretchSensor := FALSE,
    limitUnstretchSensor := FALSE,
    unstretch => P1_050_DO2.digitalOutput_04); // FB_FormingBoardWireStretchControl
P1_050_DO2.digitalOutput_03 := instFB_FormingBoardWireStretchControl.stretch;
END_METHOD

METHOD _MixPumpControl_1
VAR_INPUT
END_VAR
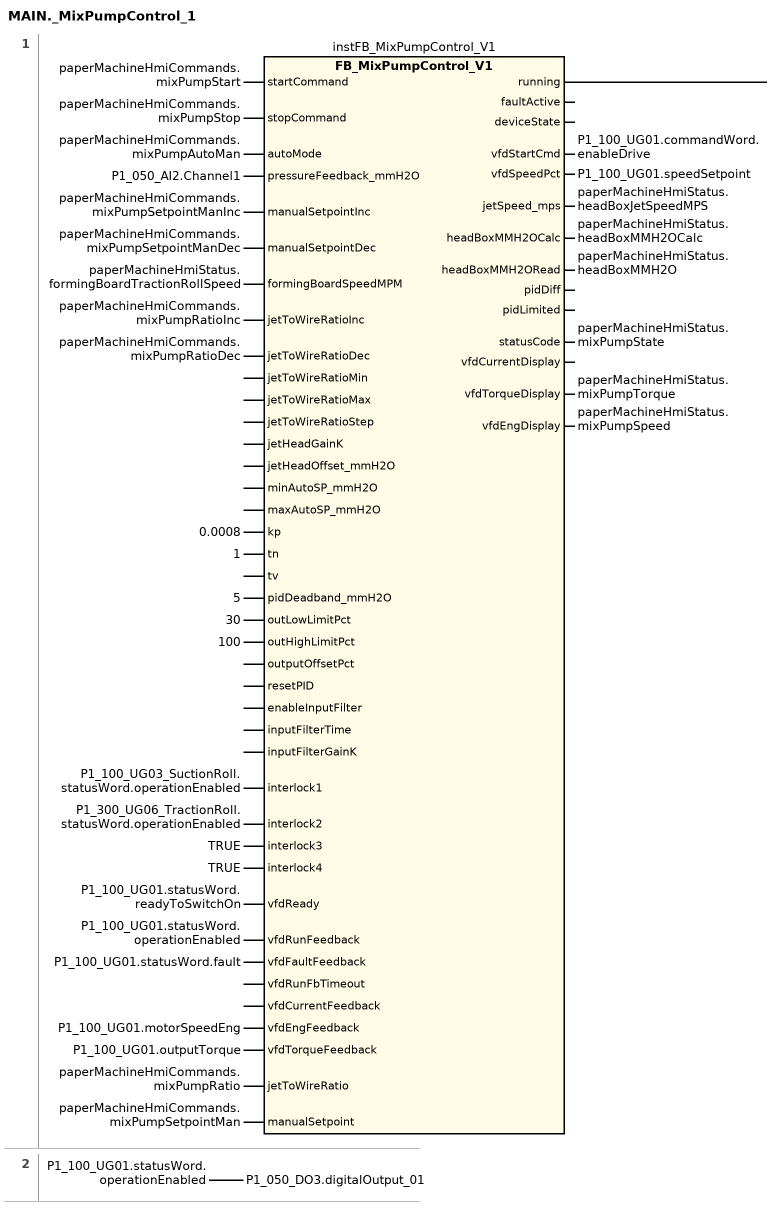
// NETWORK 1
instFB_MixPumpControl_V1(
    startCommand := paperMachineHmiCommands.mixPumpStart,
    stopCommand := paperMachineHmiCommands.mixPumpStop,
    autoMode := paperMachineHmiCommands.mixPumpAutoMan,
    pressureFeedback_mmH2O := P1_050_AI2.Channel1,
    manualSetpointInc := paperMachineHmiCommands.mixPumpSetpointManInc,
    manualSetpointDec := paperMachineHmiCommands.mixPumpSetpointManDec,
    formingBoardSpeedMPM := paperMachineHmiStatus.formingBoardTractionRollSpeed,
    jetToWireRatioInc := paperMachineHmiCommands.mixPumpRatioInc,
    jetToWireRatioDec := paperMachineHmiCommands.mixPumpRatioDec,
    kp := 0.0008,
    tn := 1,
    pidDeadband_mmH2O := 5,
    outLowLimitPct := 30,
    outHighLimitPct := 100,
    interlock1 := P1_100_UG03_SuctionRoll.statusWord.operationEnabled,
    interlock2 := P1_300_UG06_TractionRoll.statusWord.operationEnabled,
    interlock3 := TRUE,
    interlock4 := TRUE,
    vfdReady := P1_100_UG01.statusWord.readyToSwitchOn,
    vfdRunFeedback := P1_100_UG01.statusWord.operationEnabled,
    vfdFaultFeedback := P1_100_UG01.statusWord.fault,
    vfdEngFeedback := P1_100_UG01.motorSpeedEng,
    vfdTorqueFeedback := P1_100_UG01.outputTorque,
    jetToWireRatio := paperMachineHmiCommands.mixPumpRatio,
    manualSetpoint := paperMachineHmiCommands.mixPumpSetpointMan,
    vfdStartCmd => P1_100_UG01.commandWord.enableDrive,
    vfdSpeedPct => P1_100_UG01.speedSetpoint,
    jetSpeed_mps => paperMachineHmiStatus.headBoxJetSpeedMPS,
    headBoxMMH2OCalc => paperMachineHmiStatus.headBoxMMH2OCalc,
    headBoxMMH2ORead => paperMachineHmiStatus.headBoxMMH2O,
    statusCode => paperMachineHmiStatus.mixPumpState,
    vfdTorqueDisplay => paperMachineHmiStatus.mixPumpTorque,
    vfdEngDisplay => paperMachineHmiStatus.mixPumpSpeed); // FB_MixPumpControl_V1

// NETWORK 2
P1_050_DO3.digitalOutput_01 := P1_100_UG01.statusWord.operationEnabled;
END_METHOD

METHOD _StockPumpControl
VAR_INPUT
END_VAR

VAR
END_VAR
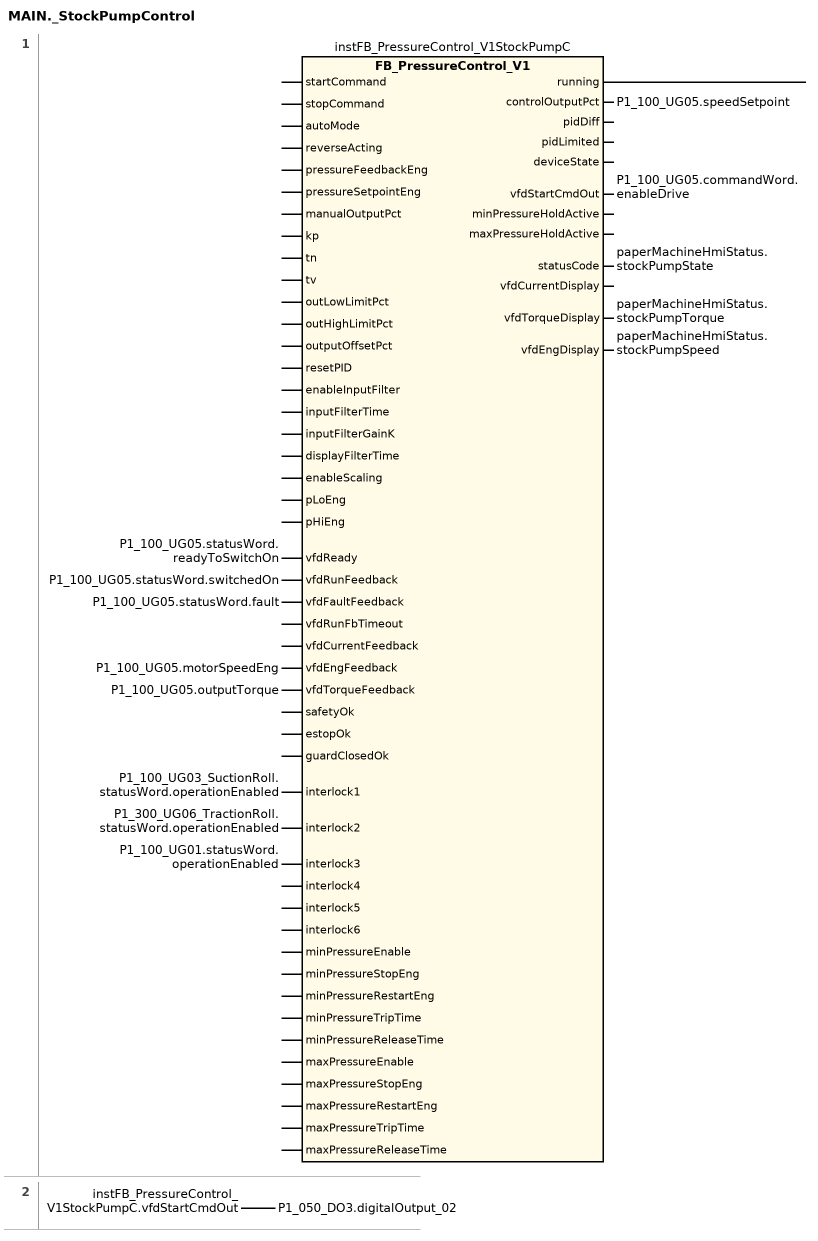
// NETWORK 1
instFB_PressureControl_V1StockPumpC(
    vfdReady := P1_100_UG05.statusWord.readyToSwitchOn,
    vfdRunFeedback := P1_100_UG05.statusWord.switchedOn,
    vfdFaultFeedback := P1_100_UG05.statusWord.fault,
    vfdEngFeedback := P1_100_UG05.motorSpeedEng,
    vfdTorqueFeedback := P1_100_UG05.outputTorque,
    interlock1 := P1_100_UG03_SuctionRoll.statusWord.operationEnabled,
    interlock2 := P1_300_UG06_TractionRoll.statusWord.operationEnabled,
    interlock3 := P1_100_UG01.statusWord.operationEnabled,
    controlOutputPct => P1_100_UG05.speedSetpoint,
    vfdStartCmdOut => P1_100_UG05.commandWord.enableDrive,
    statusCode => paperMachineHmiStatus.stockPumpState,
    vfdTorqueDisplay => paperMachineHmiStatus.stockPumpTorque,
    vfdEngDisplay => paperMachineHmiStatus.stockPumpSpeed); // FB_PressureControl_V1

// NETWORK 2
P1_050_DO3.digitalOutput_02 := instFB_PressureControl_V1StockPumpC.vfdStartCmdOut;
END_METHOD

METHOD _StockPumpControl_1
VAR_INPUT
END_VAR

VAR
END_VAR
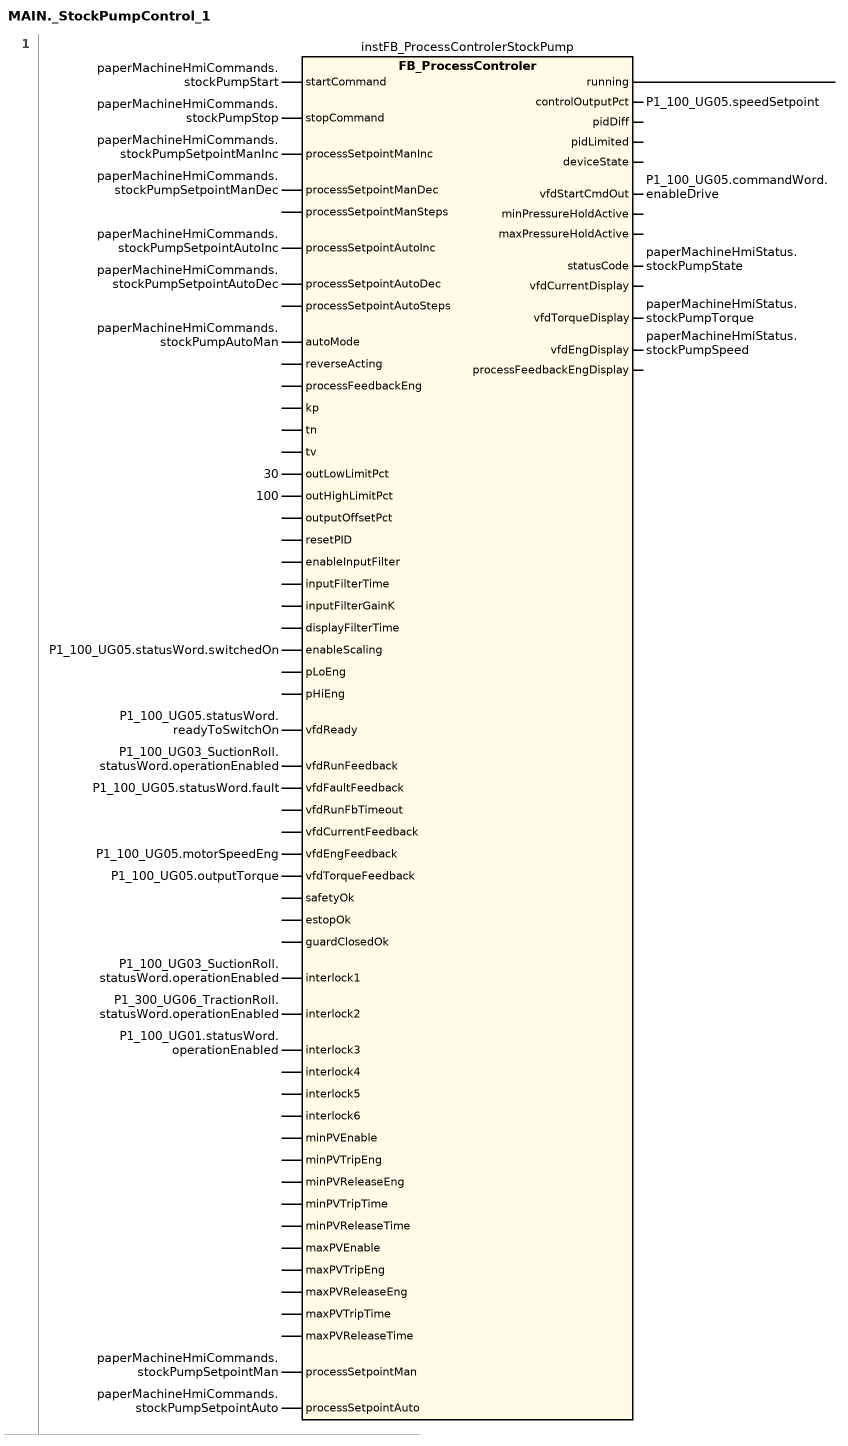
// NETWORK 1
instFB_ProcessControlerStockPump(
    startCommand := paperMachineHmiCommands.stockPumpStart,
    stopCommand := paperMachineHmiCommands.stockPumpStop,
    processSetpointManInc := paperMachineHmiCommands.stockPumpSetpointManInc,
    processSetpointManDec := paperMachineHmiCommands.stockPumpSetpointManDec,
    processSetpointAutoInc := paperMachineHmiCommands.stockPumpSetpointAutoInc,
    processSetpointAutoDec := paperMachineHmiCommands.stockPumpSetpointAutoDec,
    autoMode := paperMachineHmiCommands.stockPumpAutoMan,
    outLowLimitPct := 30,
    outHighLimitPct := 100,
    enableScaling := P1_100_UG05.statusWord.switchedOn,
    vfdReady := P1_100_UG05.statusWord.readyToSwitchOn,
    vfdRunFeedback := P1_100_UG03_SuctionRoll.statusWord.operationEnabled,
    vfdFaultFeedback := P1_100_UG05.statusWord.fault,
    vfdEngFeedback := P1_100_UG05.motorSpeedEng,
    vfdTorqueFeedback := P1_100_UG05.outputTorque,
    interlock1 := P1_100_UG03_SuctionRoll.statusWord.operationEnabled,
    interlock2 := P1_300_UG06_TractionRoll.statusWord.operationEnabled,
    interlock3 := P1_100_UG01.statusWord.operationEnabled,
    processSetpointMan := paperMachineHmiCommands.stockPumpSetpointMan,
    processSetpointAuto := paperMachineHmiCommands.stockPumpSetpointAuto,
    controlOutputPct => P1_100_UG05.speedSetpoint,
    vfdStartCmdOut => P1_100_UG05.commandWord.enableDrive,
    statusCode => paperMachineHmiStatus.stockPumpState,
    vfdTorqueDisplay => paperMachineHmiStatus.stockPumpTorque,
    vfdEngDisplay => paperMachineHmiStatus.stockPumpSpeed); // FB_ProcessControler

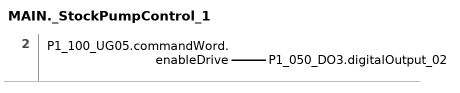
// NETWORK 2
P1_050_DO3.digitalOutput_02 := P1_100_UG05.commandWord.enableDrive;
END_METHOD

METHOD _VaccumPumps
VAR_INPUT
END_VAR
(*

    // ─────────────── LOW VACUUM EXHAUST FAN ───────────────
    lowVacuumExhaustFanStart : BOOL;  // Start low vacuum exhaust fan (Ligar exaustor do baixo vácuo)
    lowVacuumExhaustFanStop  : BOOL;  // Stop low vacuum exhaust fan (Parar exaustor do baixo vácuo)
	
	paperMachineHmiCommands.suctionRollVacuumPumpStart
	paperMachineHmiCommands.suctionRollVacuumPumpStop
	paperMachineHmiCommands.wireVacuumPumpStart
	paperMachineHmiCommands.wireVacuumPumpStop


*)
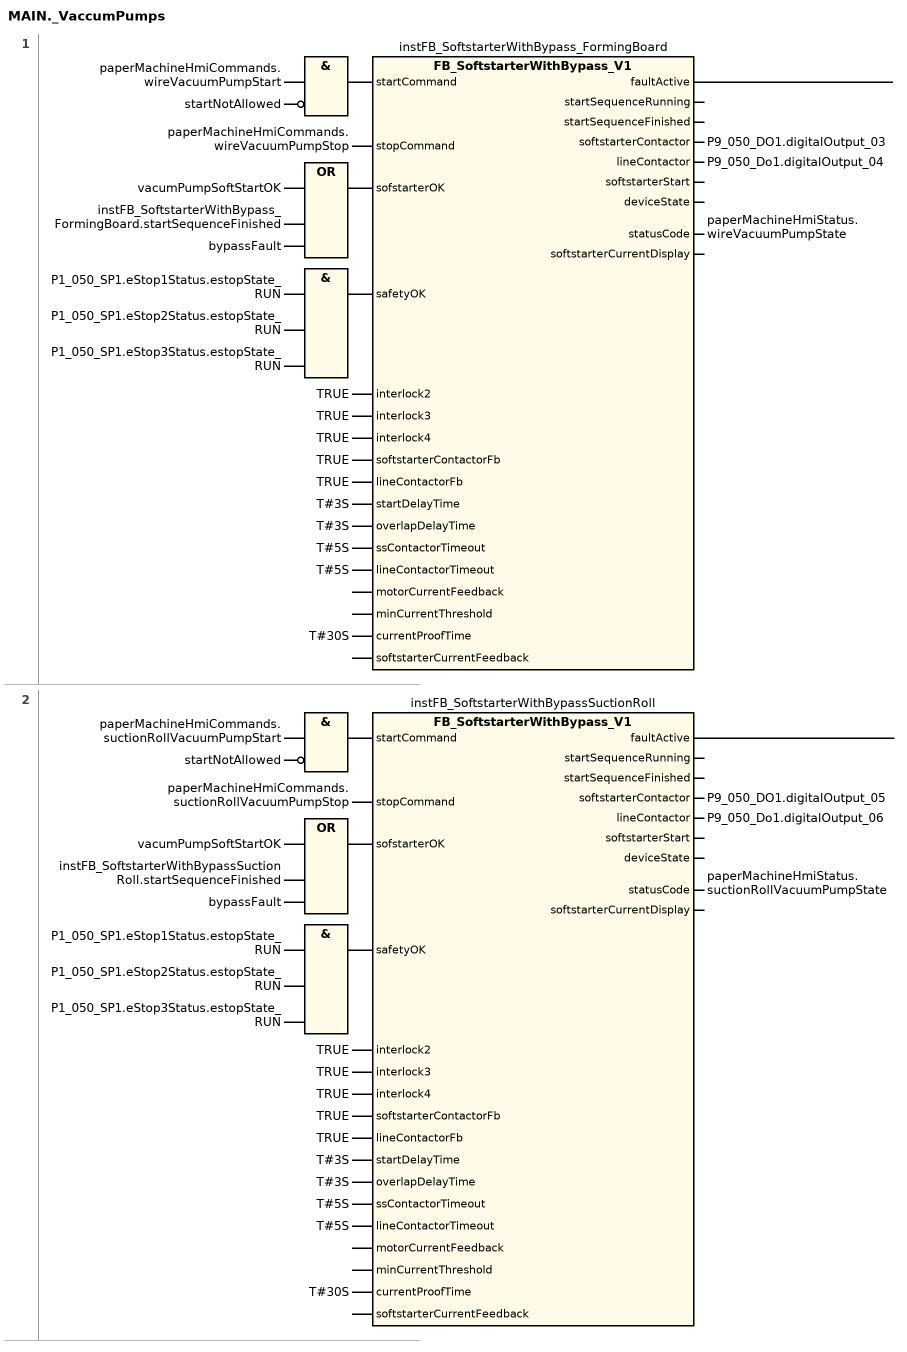
// NETWORK 1
instFB_SoftstarterWithBypass_FormingBoard(
    startCommand := paperMachineHmiCommands.wireVacuumPumpStart AND NOT startNotAllowed,
    stopCommand := paperMachineHmiCommands.wireVacuumPumpStop,
    sofstarterOK := vacumPumpSoftStartOK OR instFB_SoftstarterWithBypass_FormingBoard.startSequenceFinished OR bypassFault,
    safetyOK := P1_050_SP1.eStop1Status.estopState_RUN AND P1_050_SP1.eStop2Status.estopState_RUN AND P1_050_SP1.eStop3Status.estopState_RUN,
    interlock2 := TRUE,
    interlock3 := TRUE,
    interlock4 := TRUE,
    softstarterContactorFb := TRUE,
    lineContactorFb := TRUE,
    startDelayTime := T#3S,
    overlapDelayTime := T#3S,
    ssContactorTimeout := T#5S,
    lineContactorTimeout := T#5S,
    currentProofTime := T#30S,
    softstarterContactor => P9_050_DO1.digitalOutput_03,
    lineContactor => P9_050_Do1.digitalOutput_04,
    statusCode => paperMachineHmiStatus.wireVacuumPumpState); // FB_SoftstarterWithBypass_V1

// NETWORK 2
instFB_SoftstarterWithBypassSuctionRoll(
    startCommand := paperMachineHmiCommands.suctionRollVacuumPumpStart AND NOT startNotAllowed,
    stopCommand := paperMachineHmiCommands.suctionRollVacuumPumpStop,
    sofstarterOK := vacumPumpSoftStartOK OR instFB_SoftstarterWithBypassSuctionRoll.startSequenceFinished OR bypassFault,
    safetyOK := P1_050_SP1.eStop1Status.estopState_RUN AND P1_050_SP1.eStop2Status.estopState_RUN AND P1_050_SP1.eStop3Status.estopState_RUN,
    interlock2 := TRUE,
    interlock3 := TRUE,
    interlock4 := TRUE,
    softstarterContactorFb := TRUE,
    lineContactorFb := TRUE,
    startDelayTime := T#3S,
    overlapDelayTime := T#3S,
    ssContactorTimeout := T#5S,
    lineContactorTimeout := T#5S,
    currentProofTime := T#30S,
    softstarterContactor => P9_050_DO1.digitalOutput_05,
    lineContactor => P9_050_Do1.digitalOutput_06,
    statusCode => paperMachineHmiStatus.suctionRollVacuumPumpState); // FB_SoftstarterWithBypass_V1

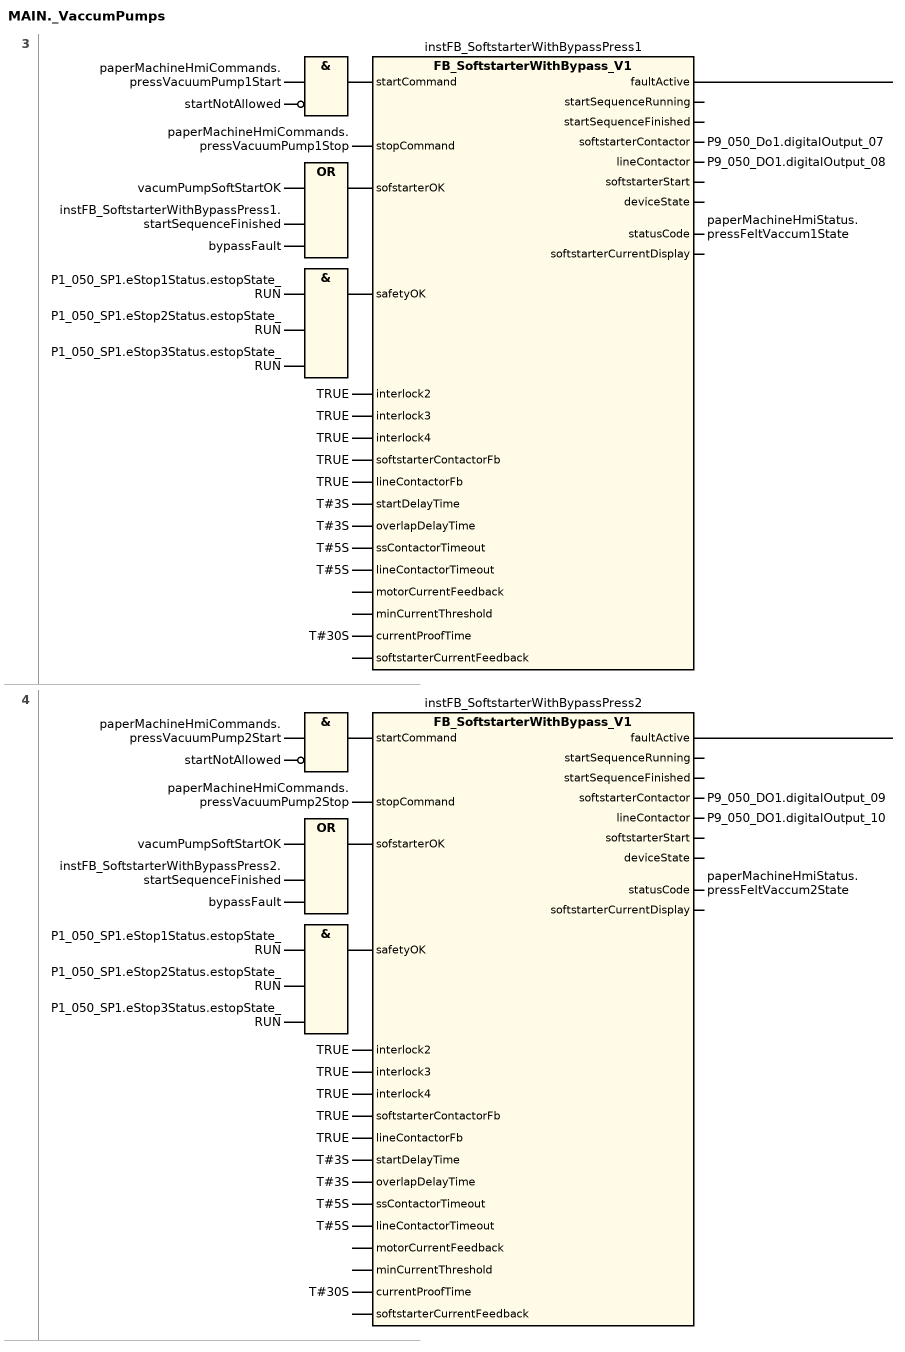
// NETWORK 3
instFB_SoftstarterWithBypassPress1(
    startCommand := paperMachineHmiCommands.pressVacuumPump1Start AND NOT startNotAllowed,
    stopCommand := paperMachineHmiCommands.pressVacuumPump1Stop,
    sofstarterOK := vacumPumpSoftStartOK OR instFB_SoftstarterWithBypassPress1.startSequenceFinished OR bypassFault,
    safetyOK := P1_050_SP1.eStop1Status.estopState_RUN AND P1_050_SP1.eStop2Status.estopState_RUN AND P1_050_SP1.eStop3Status.estopState_RUN,
    interlock2 := TRUE,
    interlock3 := TRUE,
    interlock4 := TRUE,
    softstarterContactorFb := TRUE,
    lineContactorFb := TRUE,
    startDelayTime := T#3S,
    overlapDelayTime := T#3S,
    ssContactorTimeout := T#5S,
    lineContactorTimeout := T#5S,
    currentProofTime := T#30S,
    softstarterContactor => P9_050_Do1.digitalOutput_07,
    lineContactor => P9_050_DO1.digitalOutput_08,
    statusCode => paperMachineHmiStatus.pressFeltVaccum1State); // FB_SoftstarterWithBypass_V1

// NETWORK 4
instFB_SoftstarterWithBypassPress2(
    startCommand := paperMachineHmiCommands.pressVacuumPump2Start AND NOT startNotAllowed,
    stopCommand := paperMachineHmiCommands.pressVacuumPump2Stop,
    sofstarterOK := vacumPumpSoftStartOK OR instFB_SoftstarterWithBypassPress2.startSequenceFinished OR bypassFault,
    safetyOK := P1_050_SP1.eStop1Status.estopState_RUN AND P1_050_SP1.eStop2Status.estopState_RUN AND P1_050_SP1.eStop3Status.estopState_RUN,
    interlock2 := TRUE,
    interlock3 := TRUE,
    interlock4 := TRUE,
    softstarterContactorFb := TRUE,
    lineContactorFb := TRUE,
    startDelayTime := T#3S,
    overlapDelayTime := T#3S,
    ssContactorTimeout := T#5S,
    lineContactorTimeout := T#5S,
    currentProofTime := T#30S,
    softstarterContactor => P9_050_DO1.digitalOutput_09,
    lineContactor => P9_050_DO1.digitalOutput_10,
    statusCode => paperMachineHmiStatus.pressFeltVaccum2State); // FB_SoftstarterWithBypass_V1

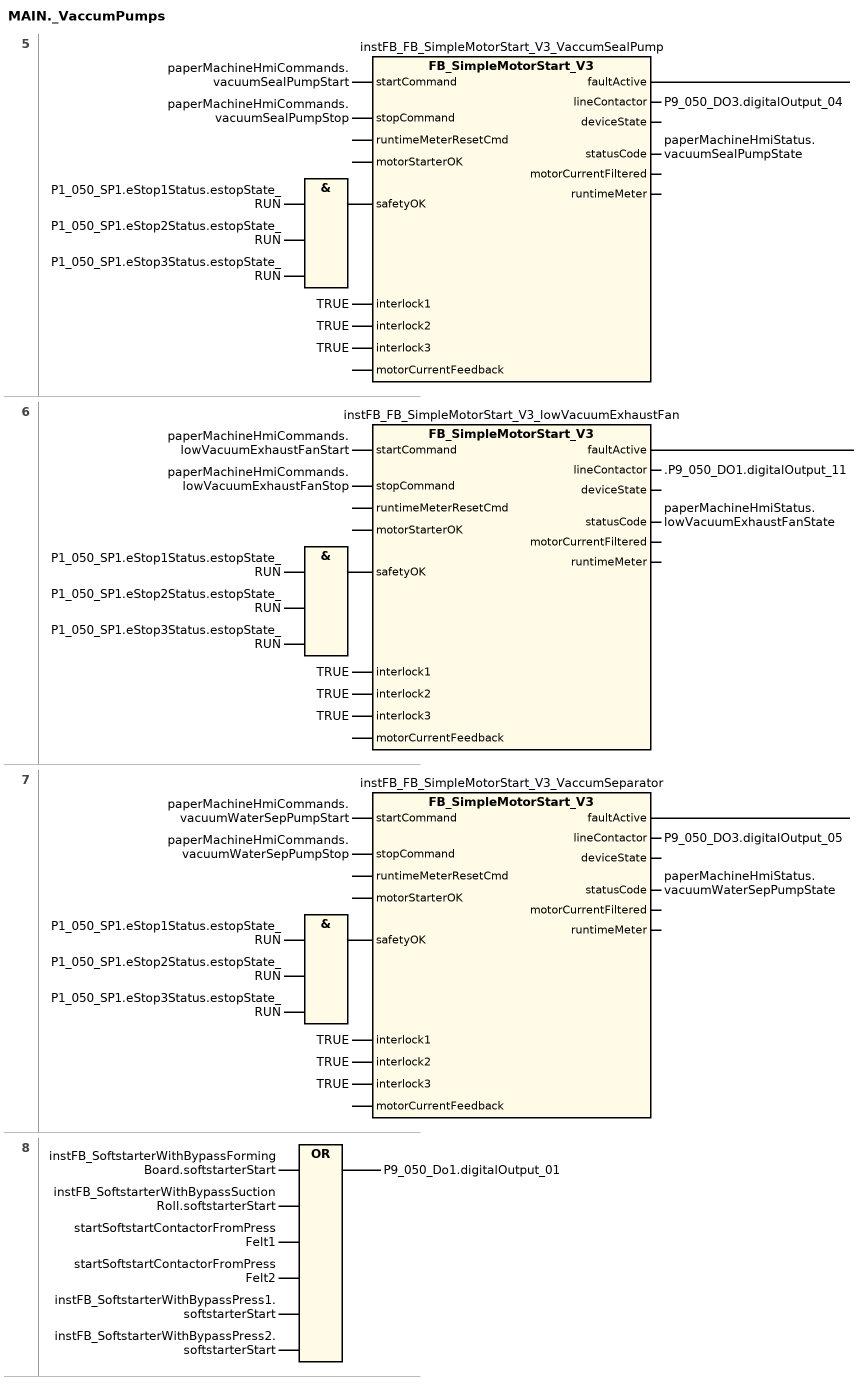
// NETWORK 5
instFB_FB_SimpleMotorStart_V3_VaccumSealPump(
    startCommand := paperMachineHmiCommands.vacuumSealPumpStart,
    stopCommand := paperMachineHmiCommands.vacuumSealPumpStop,
    safetyOK := P1_050_SP1.eStop1Status.estopState_RUN AND P1_050_SP1.eStop2Status.estopState_RUN AND P1_050_SP1.eStop3Status.estopState_RUN,
    interlock1 := TRUE,
    interlock2 := TRUE,
    interlock3 := TRUE,
    lineContactor => P9_050_DO3.digitalOutput_04,
    statusCode => paperMachineHmiStatus.vacuumSealPumpState); // FB_SimpleMotorStart_V3

// NETWORK 6
instFB_FB_SimpleMotorStart_V3_lowVacuumExhaustFan(
    startCommand := paperMachineHmiCommands.lowVacuumExhaustFanStart,
    stopCommand := paperMachineHmiCommands.lowVacuumExhaustFanStop,
    safetyOK := P1_050_SP1.eStop1Status.estopState_RUN AND P1_050_SP1.eStop2Status.estopState_RUN AND P1_050_SP1.eStop3Status.estopState_RUN,
    interlock1 := TRUE,
    interlock2 := TRUE,
    interlock3 := TRUE,
    lineContactor => .P9_050_DO1.digitalOutput_11,
    statusCode => paperMachineHmiStatus.lowVacuumExhaustFanState); // FB_SimpleMotorStart_V3

// NETWORK 7
instFB_FB_SimpleMotorStart_V3_VaccumSeparator(
    startCommand := paperMachineHmiCommands.vacuumWaterSepPumpStart,
    stopCommand := paperMachineHmiCommands.vacuumWaterSepPumpStop,
    safetyOK := P1_050_SP1.eStop1Status.estopState_RUN AND P1_050_SP1.eStop2Status.estopState_RUN AND P1_050_SP1.eStop3Status.estopState_RUN,
    interlock1 := TRUE,
    interlock2 := TRUE,
    interlock3 := TRUE,
    lineContactor => P9_050_DO3.digitalOutput_05,
    statusCode => paperMachineHmiStatus.vacuumWaterSepPumpState); // FB_SimpleMotorStart_V3

// NETWORK 8
P9_050_Do1.digitalOutput_01 := instFB_SoftstarterWithBypassFormingBoard.softstarterStart OR instFB_SoftstarterWithBypassSuctionRoll.softstarterStart OR startSoftstartContactorFromPressFelt1 OR startSoftstartContactorFromPressFelt2 OR instFB_SoftstarterWithBypassPress1.softstarterStart OR instFB_SoftstarterWithBypassPress2.softstarterStart;

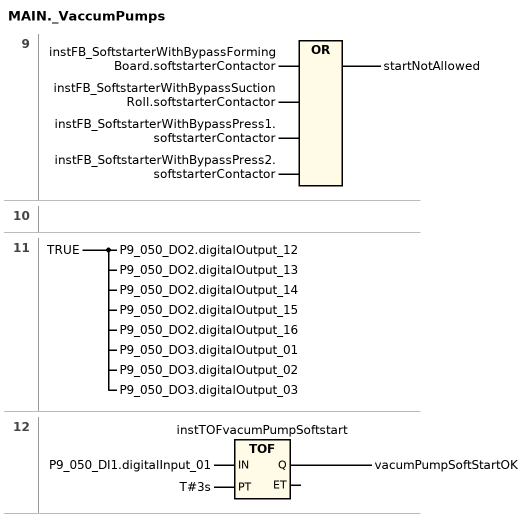
// NETWORK 9
startNotAllowed := instFB_SoftstarterWithBypassFormingBoard.softstarterContactor OR instFB_SoftstarterWithBypassSuctionRoll.softstarterContactor OR instFB_SoftstarterWithBypassPress1.softstarterContactor OR instFB_SoftstarterWithBypassPress2.softstarterContactor;

// NETWORK 10

// NETWORK 11
P9_050_DO2.digitalOutput_12 := TRUE;
P9_050_DO2.digitalOutput_13 := TRUE;
P9_050_DO2.digitalOutput_14 := TRUE;
P9_050_DO2.digitalOutput_15 := TRUE;
P9_050_DO2.digitalOutput_16 := TRUE;
P9_050_DO3.digitalOutput_01 := TRUE;
P9_050_DO3.digitalOutput_02 := TRUE;
P9_050_DO3.digitalOutput_03 := TRUE;

// NETWORK 12
instTOFvacumPumpSoftstart(IN := P9_050_DI1.digitalInput_01, PT := T#3s); // TOF
vacumPumpSoftStartOK := instTOFvacumPumpSoftstart.Q;
END_METHOD

METHOD _WirePitPumpControl
VAR_INPUT
END_VAR
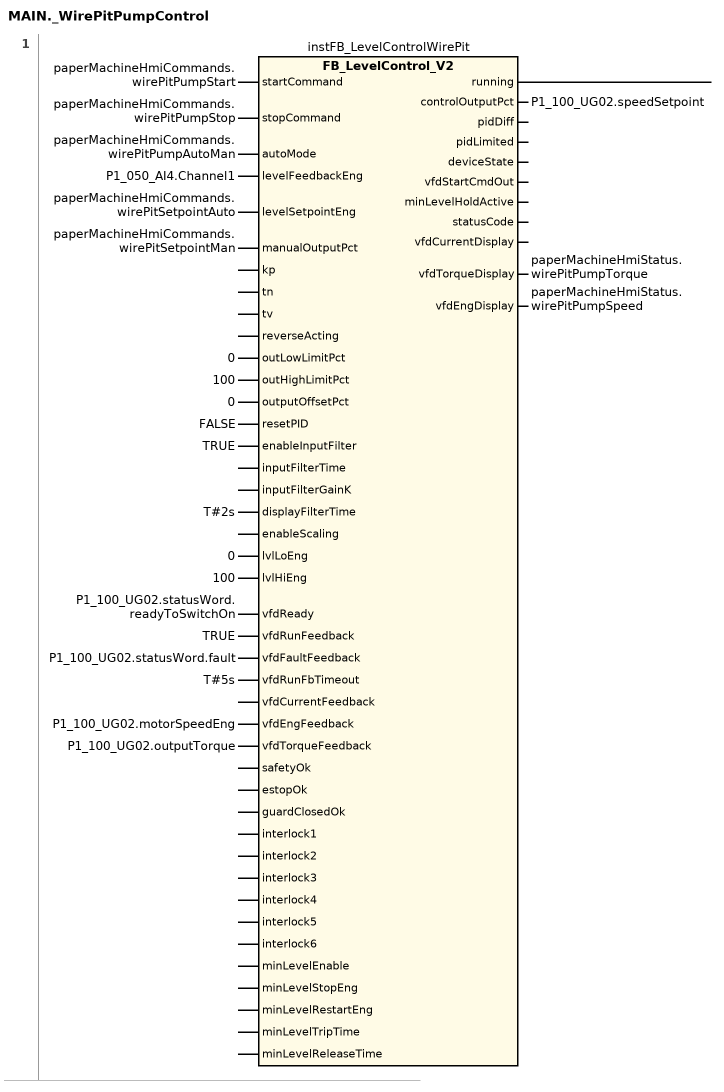
// NETWORK 1
instFB_LevelControlWirePit(
    startCommand := paperMachineHmiCommands.wirePitPumpStart,
    stopCommand := paperMachineHmiCommands.wirePitPumpStop,
    autoMode := paperMachineHmiCommands.wirePitPumpAutoMan,
    levelFeedbackEng := P1_050_AI4.Channel1,
    levelSetpointEng := paperMachineHmiCommands.wirePitSetpointAuto,
    manualOutputPct := paperMachineHmiCommands.wirePitSetpointMan,
    outLowLimitPct := 0,
    outHighLimitPct := 100,
    outputOffsetPct := 0,
    resetPID := FALSE,
    enableInputFilter := TRUE,
    displayFilterTime := T#2s,
    lvlLoEng := 0,
    lvlHiEng := 100,
    vfdReady := P1_100_UG02.statusWord.readyToSwitchOn,
    vfdRunFeedback := TRUE,
    vfdFaultFeedback := P1_100_UG02.statusWord.fault,
    vfdRunFbTimeout := T#5s,
    vfdEngFeedback := P1_100_UG02.motorSpeedEng,
    vfdTorqueFeedback := P1_100_UG02.outputTorque,
    controlOutputPct => P1_100_UG02.speedSetpoint,
    vfdTorqueDisplay => paperMachineHmiStatus.wirePitPumpTorque,
    vfdEngDisplay => paperMachineHmiStatus.wirePitPumpSpeed); // FB_LevelControl_V2
END_METHOD

METHOD _WirePitPumpControl_1
VAR_INPUT
END_VAR
